C01814=1060.233,-44.337,-65.681,171.446,27.282,155.095
C01815=1060.228,-44.587,-65.669,171.444,27.280,155.095
C01816=1060.221,-44.836,-65.657,171.442,27.279,155.095
C01817=1060.215,-45.086,-65.644,171.441,27.277,155.095
C01818=1060.209,-45.335,-65.631,171.439,27.275,155.095
C01819=1060.203,-45.585,-65.619,171.437,27.273,155.094
C01820=1060.196,-45.835,-65.607,171.436,27.271,155.094
C01821=1060.190,-46.085,-65.594,171.434,27.269,155.094
C01822=1060.184,-46.335,-65.581,171.432,27.267,155.094
C01823=1060.178,-46.584,-65.568,171.431,27.265,155.094
C01824=1060.172,-46.833,-65.556,171.429,27.263,155.093
C01825=1060.166,-47.083,-65.544,171.428,27.261,155.093
C01826=1060.160,-47.332,-65.531,171.426,27.259,155.093
C01827=1060.154,-47.582,-65.519,171.424,27.257,155.093
C01828=1060.147,-47.831,-65.506,171.423,27.255,155.093
C01829=1060.142,-48.081,-65.494,171.421,27.254,155.093
C01830=1060.136,-48.331,-65.481,171.419,27.251,155.092
C01831=1060.130,-48.581,-65.469,171.418,27.250,155.092
C01832=1060.123,-48.831,-65.457,171.416,27.247,155.092
C01833=1060.117,-49.080,-65.444,171.414,27.246,155.092
C01834=1060.112,-49.330,-65.432,171.413,27.244,155.092
C01835=1060.105,-49.579,-65.419,171.411,27.242,155.091
C01836=1060.099,-49.828,-65.407,171.409,27.240,155.091
C01837=1060.093,-50.108,-65.393,171.408,27.238,155.091
C01838=1060.086,-50.387,-65.379,171.406,27.236,155.091
C01839=1060.078,-50.667,-65.365,171.403,27.234,155.091
C01840=1060.071,-50.946,-65.352,171.402,27.232,155.091
C01841=1060.065,-51.195,-65.340,171.400,27.230,155.090
C01842=1060.059,-51.444,-65.327,171.399,27.228,155.090
C01843=1060.053,-51.694,-65.315,171.397,27.227,155.090
C01844=1060.047,-51.944,-65.303,171.395,27.225,155.090
C01845=1060.040,-52.193,-65.291,171.394,27.223,155.090
C01846=1060.034,-52.443,-65.278,171.392,27.221,155.090
C01847=1060.028,-52.693,-65.266,171.390,27.219,155.089
C01848=1060.021,-52.942,-65.254,171.389,27.218,155.089
C01849=1060.015,-53.192,-65.242,171.387,27.216,155.089
C01850=1060.008,-53.442,-65.230,171.385,27.214,155.089
C01851=1060.003,-53.691,-65.218,171.384,27.213,155.089
C01852=1059.996,-53.941,-65.206,171.382,27.211,155.089
C01853=1059.990,-54.190,-65.194,171.380,27.209,155.089
C01854=1059.984,-54.440,-65.181,171.378,27.207,155.088
C01855=1059.977,-54.690,-65.169,171.377,27.206,155.088
C01856=1059.971,-54.940,-65.157,171.375,27.203,155.088
C01857=1059.965,-55.189,-65.145,171.374,27.202,155.088
C01858=1059.959,-55.438,-65.133,171.371,27.200,155.088
C01859=1059.953,-55.688,-65.121,171.369,27.198,155.088
C01860=1059.946,-55.938,-65.109,171.368,27.196,155.087
C01861=1059.940,-56.188,-65.097,171.366,27.195,155.087
C01862=1059.934,-56.437,-65.085,171.364,27.193,155.087
C01863=1059.928,-56.686,-65.073,171.362,27.191,155.087
C01864=1059.922,-56.936,-65.061,171.361,27.190,155.087
C01865=1059.915,-57.186,-65.049,171.359,27.188,155.087
C01866=1059.909,-57.435,-65.037,171.357,27.186,155.087
C01867=1059.903,-57.686,-65.025,171.356,27.184,155.086
C01868=1059.897,-57.935,-65.013,171.354,27.183,155.086
C01869=1059.890,-58.184,-65.001,171.352,27.181,155.086
C01870=1059.884,-58.434,-64.989,171.351,27.179,155.086
C01871=1059.878,-58.684,-64.977,171.349,27.178,155.086
C01872=1059.872,-58.933,-64.966,171.347,27.176,155.086
C01873=1059.866,-59.183,-64.953,171.346,27.174,155.086
C01874=1059.859,-59.433,-64.942,171.344,27.172,155.085
C01875=1059.853,-59.682,-64.930,171.342,27.171,155.085
C01876=1059.847,-59.931,-64.917,171.341,27.169,155.085
C01877=1059.841,-60.182,-64.906,171.339,27.167,155.085
C01878=1059.834,-60.431,-64.894,171.337,27.166,155.085
C01879=1059.829,-60.681,-64.882,171.336,27.164,155.085
C01880=1059.823,-60.930,-64.870,171.334,27.162,155.085
C01881=1059.816,-61.180,-64.859,171.332,27.161,155.084
C01882=1059.810,-61.430,-64.846,171.331,27.159,155.084
C01883=1059.804,-61.680,-64.834,171.329,27.157,155.084
C01884=1059.798,-61.929,-64.823,171.326,27.155,155.084
C01885=1059.792,-62.179,-64.811,171.325,27.153,155.084
C01886=1059.785,-62.429,-64.799,171.323,27.152,155.084
C01887=1059.779,-62.677,-64.787,171.321,27.150,155.084
C01888=1059.774,-62.928,-64.775,171.320,27.148,155.083
C01889=1059.767,-63.178,-64.763,171.318,27.147,155.083
C01890=1059.761,-63.426,-64.752,171.316,27.145,155.083
C01891=1059.755,-63.677,-64.740,171.315,27.143,155.083
C01892=1059.749,-63.926,-64.728,171.313,27.141,155.083
C01893=1059.743,-64.175,-64.717,171.311,27.140,155.083
C01894=1059.736,-64.426,-64.705,171.309,27.138,155.083
C01895=1059.730,-64.675,-64.693,171.308,27.136,155.082
C01896=1059.725,-64.925,-64.682,171.306,27.135,155.082
C01897=1059.718,-65.174,-64.670,171.304,27.134,155.082
C01898=1059.712,-65.424,-64.657,171.303,27.132,155.082
C01899=1059.706,-65.674,-64.646,171.301,27.130,155.082
C01900=1059.700,-65.923,-64.634,171.299,27.128,155.082
C01901=1059.693,-66.204,-64.622,171.297,27.126,155.082
C01902=1059.686,-66.484,-64.608,171.295,27.125,155.082
C01903=1059.680,-66.765,-64.596,171.293,27.123,155.081
C01904=1059.672,-67.045,-64.582,171.292,27.121,155.081
C01905=1059.667,-67.295,-64.571,171.290,27.120,155.081
C01906=1059.661,-67.545,-64.559,171.287,27.118,155.081
C01907=1059.654,-67.794,-64.547,171.286,27.116,155.081
C01908=1059.648,-68.044,-64.536,171.284,27.114,155.081
C01909=1059.642,-68.293,-64.523,171.282,27.112,155.081
C01910=1059.637,-68.543,-64.512,171.281,27.111,155.080
C01911=1059.630,-68.793,-64.501,171.279,27.109,155.080
C01912=1059.624,-69.042,-64.490,171.277,27.107,155.080
C01913=1059.618,-69.292,-64.477,171.276,27.106,155.080
C01914=1059.612,-69.542,-64.466,171.274,27.104,155.080
C01915=1059.606,-69.791,-64.454,171.272,27.103,155.080
C01916=1059.600,-70.041,-64.443,171.270,27.101,155.080
C01917=1059.594,-70.291,-64.432,171.269,27.099,155.080
C01918=1059.588,-70.541,-64.420,171.267,27.098,155.079
C01919=1059.582,-70.790,-64.409,171.265,27.097,155.079
C01920=1059.576,-71.040,-64.397,171.264,27.095,155.079
C01921=1059.570,-71.289,-64.386,171.262,27.093,155.079
C01922=1059.564,-71.539,-64.373,171.260,27.091,155.079
C01923=1059.558,-71.788,-64.362,171.259,27.090,155.079
C01924=1059.552,-72.039,-64.351,171.257,27.089,155.079
C01925=1059.546,-72.288,-64.340,171.255,27.087,155.079
C01926=1059.539,-72.538,-64.328,171.253,27.085,155.079
C01927=1059.534,-72.787,-64.316,171.251,27.083,155.078
C01928=1059.528,-73.037,-64.305,171.249,27.082,155.078
C01929=1059.522,-73.287,-64.294,171.247,27.080,155.078
C01930=1059.515,-73.536,-64.282,171.246,27.079,155.078
C01931=1059.510,-73.786,-64.271,171.244,27.077,155.078
C01932=1059.504,-74.036,-64.259,171.242,27.076,155.078
C01933=1059.497,-74.285,-64.248,171.241,27.074,155.078
C01934=1059.491,-74.535,-64.237,171.239,27.072,155.078
C01935=1059.485,-74.784,-64.226,171.237,27.071,155.078
C01936=1059.479,-75.034,-64.214,171.235,27.070,155.078
C01937=1059.473,-75.283,-64.203,171.234,27.068,155.077
C01938=1059.467,-75.534,-64.192,171.232,27.067,155.077
C01939=1059.461,-75.783,-64.181,171.230,27.065,155.077
C01940=1059.454,-76.033,-64.169,171.229,27.064,155.077
C01941=1059.448,-76.282,-64.158,171.227,27.062,155.077
C01942=1059.442,-76.532,-64.147,171.225,27.061,155.077
C01943=1059.436,-76.782,-64.136,171.223,27.059,155.077
C01944=1059.430,-77.031,-64.124,171.221,27.057,155.077
C01945=1059.424,-77.281,-64.113,171.219,27.056,155.077
C01946=1059.418,-77.531,-64.102,171.217,27.054,155.077
C01947=1059.412,-77.781,-64.091,171.216,27.053,155.077
C01948=1059.406,-78.031,-64.080,171.214,27.052,155.076
C01949=1059.399,-78.280,-64.069,171.212,27.051,155.076
C01950=1059.393,-78.530,-64.057,171.210,27.049,155.076
C01951=1059.387,-78.779,-64.046,171.209,27.048,155.076
C01952=1059.381,-79.030,-64.035,171.207,27.046,155.076
C01953=1059.375,-79.279,-64.024,171.205,27.045,155.076
C01954=1059.369,-79.528,-64.013,171.204,27.043,155.076
C01955=1059.363,-79.778,-64.001,171.202,27.042,155.076
C01956=1059.356,-80.027,-63.991,171.200,27.040,155.076
C01957=1059.350,-80.277,-63.980,171.198,27.039,155.076
C01958=1059.344,-80.527,-63.969,171.196,27.037,155.076
C01959=1059.338,-80.777,-63.958,171.194,27.036,155.076
C01960=1059.332,-81.026,-63.948,171.192,27.035,155.076
C01961=1059.325,-81.277,-63.936,171.191,27.033,155.075
C01962=1059.319,-81.526,-63.925,171.189,27.032,155.075
C01963=1059.312,-81.776,-63.915,171.187,27.031,155.075
C01964=1059.306,-82.025,-63.903,171.185,27.029,155.075
C01965=1059.300,-82.308,-63.891,171.183,27.028,155.075
C01966=1059.292,-82.590,-63.878,171.181,27.026,155.075
C01967=1059.285,-82.873,-63.867,171.179,27.025,155.075
C01968=1059.279,-83.156,-63.854,171.177,27.023,155.075
C01969=1059.272,-83.405,-63.844,171.176,27.022,155.075
C01970=1059.266,-83.655,-63.832,171.173,27.021,155.075
C01971=1059.260,-83.905,-63.821,171.171,27.019,155.075
C01972=1059.254,-84.154,-63.811,171.169,27.018,155.075
C01973=1059.247,-84.404,-63.800,171.168,27.017,155.075
C01974=1059.241,-84.654,-63.789,171.166,27.015,155.075
C01975=1059.235,-84.904,-63.778,171.164,27.014,155.075
C01976=1059.229,-85.153,-63.767,171.162,27.013,155.075
C01977=1059.223,-85.403,-63.757,171.161,27.012,155.075
C01978=1059.216,-85.653,-63.745,171.159,27.010,155.074
C01979=1059.210,-85.902,-63.735,171.157,27.009,155.074
C01980=1059.204,-86.152,-63.724,171.155,27.008,155.074
C01981=1059.198,-86.402,-63.713,171.154,27.007,155.074
C01982=1059.191,-86.651,-63.703,171.152,27.005,155.074
C01983=1059.185,-86.901,-63.691,171.149,27.004,155.074
C01984=1059.179,-87.151,-63.681,171.148,27.002,155.074
C01985=1059.173,-87.400,-63.670,171.146,27.001,155.074
C01986=1059.167,-87.651,-63.660,171.144,27.000,155.074
C01987=1059.161,-87.900,-63.649,171.142,26.998,155.074
C01988=1059.155,-88.149,-63.639,171.141,26.997,155.074
C01989=1059.148,-88.399,-63.627,171.139,26.996,155.074
C01990=1059.143,-88.649,-63.616,171.137,26.994,155.074
C01991=1059.136,-88.898,-63.606,171.135,26.993,155.074
C01992=1059.130,-89.148,-63.595,171.134,26.992,155.074
C01993=1059.124,-89.398,-63.585,171.132,26.991,155.074
C01994=1059.118,-89.648,-63.574,171.130,26.990,155.074
C01995=1059.112,-89.897,-63.564,171.128,26.989,155.074
C01996=1059.106,-90.147,-63.552,171.126,26.987,155.074
C01997=1059.099,-90.396,-63.542,171.124,26.986,155.074
C01998=1059.094,-90.646,-63.531,171.122,26.985,155.074
C01999=1059.087,-90.896,-63.521,171.120,26.983,155.074
C02000=1059.081,-91.146,-63.510,171.118,26.982,155.074
C02001=1059.075,-91.395,-63.500,171.117,26.981,155.074
C02002=1059.069,-91.645,-63.489,171.115,26.980,155.073
C02003=1059.063,-91.895,-63.479,171.113,26.978,155.073
C02004=1059.057,-92.145,-63.468,171.111,26.977,155.073
C02005=1059.051,-92.394,-63.458,171.110,26.976,155.073
C02006=1059.045,-92.644,-63.447,171.108,26.975,155.073
C02007=1059.038,-92.894,-63.437,171.106,26.974,155.073
C02008=1059.032,-93.144,-63.426,171.104,26.973,155.073
C02009=1059.027,-93.393,-63.415,171.102,26.971,155.073
C02010=1059.020,-93.642,-63.405,171.100,26.970,155.073
C02011=1059.014,-93.893,-63.394,171.098,26.969,155.073
C02012=1059.008,-94.142,-63.384,171.096,26.967,155.073
C02013=1059.002,-94.392,-63.373,171.095,26.966,155.073
C02014=1058.996,-94.642,-63.363,171.093,26.965,155.073
C02015=1058.990,-94.891,-63.353,171.091,26.964,155.073
C02016=1058.984,-95.141,-63.341,171.089,26.963,155.073
C02017=1058.977,-95.391,-63.332,171.088,26.962,155.073
C02018=1058.972,-95.640,-63.321,171.086,26.961,155.073
C02019=1058.966,-95.890,-63.310,171.084,26.959,155.073
C02020=1058.960,-96.140,-63.300,171.082,26.958,155.073
C02021=1058.954,-96.389,-63.290,171.079,26.957,155.073
C02022=1058.947,-96.639,-63.279,171.078,26.956,155.073
C02023=1058.942,-96.889,-63.269,171.076,26.955,155.073
C02024=1058.935,-97.138,-63.258,171.074,26.954,155.073
C02025=1058.930,-97.388,-63.248,171.072,26.952,155.073
C02026=1058.923,-97.638,-63.238,171.071,26.951,155.073
C02027=1058.917,-97.887,-63.227,171.069,26.950,155.073
C02028=1058.911,-98.138,-63.217,171.067,26.949,155.073
C02029=1058.904,-98.422,-63.205,171.065,26.948,155.073
C02030=1058.897,-98.707,-63.193,171.063,26.947,155.073
C02031=1058.889,-98.993,-63.182,171.061,26.945,155.073
C02032=1058.883,-99.277,-63.170,171.058,26.944,155.073
C02033=1058.876,-99.526,-63.160,171.056,26.943,155.073
C02034=1058.871,-99.777,-63.150,171.055,26.942,155.073
C02035=1058.864,-100.026,-63.140,171.053,26.941,155.073
C02036=1058.858,-100.276,-63.130,171.051,26.939,155.073
C02037=1058.852,-100.526,-63.119,171.049,26.939,155.073
C02038=1058.846,-100.776,-63.109,171.047,26.938,155.073
C02039=1058.839,-101.025,-63.099,171.046,26.937,155.073
C02040=1058.834,-101.275,-63.089,171.044,26.936,155.073
C02041=1058.827,-101.524,-63.079,171.042,26.934,155.073
C02042=1058.821,-101.774,-63.069,171.040,26.934,155.073
C02043=1058.815,-102.025,-63.058,171.037,26.933,155.073
C02044=1058.809,-102.274,-63.048,171.036,26.931,155.073
C02045=1058.802,-102.524,-63.039,171.034,26.930,155.073
C02046=1058.797,-102.773,-63.028,171.032,26.929,155.073
C02047=1058.790,-103.023,-63.018,171.030,26.929,155.073
C02048=1058.784,-103.272,-63.008,171.028,26.927,155.073
C02049=1058.779,-103.522,-62.998,171.027,26.926,155.073
C02050=1058.772,-103.772,-62.988,171.025,26.925,155.073
C02051=1058.766,-104.021,-62.978,171.023,26.925,155.073
C02052=1058.760,-104.272,-62.967,171.021,26.924,155.073
C02053=1058.754,-104.522,-62.958,171.019,26.922,155.073
C02054=1058.747,-104.771,-62.948,171.018,26.922,155.073
C02055=1058.741,-105.021,-62.938,171.015,26.920,155.073
C02056=1058.735,-105.270,-62.927,171.013,26.919,155.073
C02057=1058.729,-105.520,-62.918,171.011,26.918,155.073
C02058=1058.723,-105.770,-62.908,171.009,26.918,155.073
C02059=1058.716,-106.019,-62.898,171.008,26.917,155.073
C02060=1058.711,-106.269,-62.887,171.006,26.915,155.073
C02061=1058.705,-106.519,-62.878,171.004,26.915,155.073
C02062=1058.699,-106.769,-62.868,171.002,26.914,155.073
C02063=1058.692,-107.018,-62.858,171.000,26.913,155.073
C02064=1058.687,-107.268,-62.848,170.999,26.912,155.073
C02065=1058.681,-107.518,-62.838,170.997,26.911,155.073
C02066=1058.674,-107.767,-62.828,170.994,26.910,155.073
C02067=1058.668,-108.017,-62.818,170.992,26.909,155.073
C02068=1058.661,-108.267,-62.809,170.990,26.908,155.073
C02069=1058.655,-108.517,-62.799,170.989,26.907,155.073
C02070=1058.649,-108.766,-62.789,170.987,26.906,155.073
C02071=1058.643,-109.016,-62.779,170.985,26.906,155.073
C02072=1058.637,-109.266,-62.769,170.983,26.905,155.073
C02073=1058.631,-109.516,-62.759,170.981,26.904,155.073
C02074=1058.625,-109.766,-62.750,170.979,26.903,155.073
C02075=1058.618,-110.015,-62.740,170.978,26.902,155.074
C02076=1058.612,-110.265,-62.730,170.976,26.901,155.073
C02077=1058.606,-110.514,-62.720,170.973,26.900,155.074
C02078=1058.600,-110.764,-62.711,170.971,26.899,155.074
C02079=1058.594,-111.014,-62.701,170.969,26.899,155.074
C02080=1058.588,-111.264,-62.691,170.968,26.898,155.074
C02081=1058.582,-111.513,-62.681,170.966,26.897,155.074
C02082=1058.575,-111.763,-62.671,170.964,26.896,155.074
C02083=1058.569,-112.013,-62.662,170.962,26.895,155.074
C02084=1058.563,-112.263,-62.652,170.960,26.894,155.074
C02085=1058.557,-112.513,-62.643,170.958,26.894,155.074
C02086=1058.551,-112.762,-62.633,170.957,26.893,155.074
C02087=1058.544,-113.012,-62.623,170.955,26.892,155.074
C02088=1058.538,-113.262,-62.614,170.953,26.891,155.074
C02089=1058.532,-113.511,-62.604,170.950,26.890,155.074
C02090=1058.526,-113.761,-62.593,170.948,26.890,155.074
C02091=1058.520,-114.011,-62.584,170.946,26.889,155.074
C02092=1058.515,-114.260,-62.575,170.945,26.888,155.074
C02093=1058.507,-114.543,-62.564,170.943,26.887,155.074
C02094=1058.500,-114.827,-62.553,170.940,26.886,155.074
C02095=1058.493,-115.111,-62.542,170.938,26.886,155.075
C02096=1058.486,-115.394,-62.531,170.936,26.884,155.074
C02097=1058.480,-115.644,-62.522,170.934,26.884,155.075
C02098=1058.474,-115.894,-62.512,170.933,26.883,155.075
C02099=1058.468,-116.144,-62.503,170.930,26.882,155.075
C02100=1058.462,-116.393,-62.493,170.928,26.881,155.075
C02101=1058.456,-116.643,-62.484,170.926,26.881,155.075
C02102=1058.450,-116.892,-62.474,170.924,26.880,155.075
C02103=1058.443,-117.142,-62.465,170.922,26.879,155.075
C02104=1058.437,-117.392,-62.456,170.920,26.879,155.075
C02105=1058.431,-117.641,-62.446,170.919,26.878,155.075
C02106=1058.425,-117.891,-62.437,170.917,26.877,155.075
C02107=1058.418,-118.141,-62.427,170.915,26.876,155.075
C02108=1058.412,-118.391,-62.418,170.913,26.876,155.075
C02109=1058.406,-118.641,-62.408,170.911,26.875,155.075
C02110=1058.400,-118.890,-62.398,170.908,26.874,155.075
C02111=1058.394,-119.140,-62.389,170.907,26.873,155.076
C02112=1058.388,-119.390,-62.379,170.905,26.873,155.076
C02113=1058.382,-119.639,-62.370,170.903,26.872,155.076
C02114=1058.376,-119.889,-62.361,170.901,26.871,155.076
C02115=1058.369,-120.139,-62.352,170.899,26.871,155.076
C02116=1058.363,-120.389,-62.343,170.897,26.870,155.076
C02117=1058.357,-120.639,-62.333,170.895,26.870,155.076
C02118=1058.351,-120.888,-62.324,170.894,26.868,155.076
C02119=1058.345,-121.138,-62.314,170.892,26.868,155.076
C02120=1058.339,-121.387,-62.305,170.890,26.867,155.076
C02121=1058.333,-121.637,-62.295,170.888,26.867,155.076
C02122=1058.327,-121.888,-62.286,170.885,26.866,155.076
C02123=1058.320,-122.137,-62.277,170.883,26.866,155.077
C02124=1058.314,-122.387,-62.268,170.881,26.865,155.077
C02125=1058.308,-122.637,-62.258,170.880,26.864,155.077
C02126=1058.302,-122.886,-62.249,170.878,26.863,155.077
C02127=1058.296,-123.136,-62.240,170.876,26.863,155.077
C02128=1058.290,-123.386,-62.231,170.874,26.862,155.077
C02129=1058.283,-123.635,-62.222,170.872,26.862,155.077
C02130=1058.277,-123.885,-62.212,170.870,26.861,155.077
C02131=1058.271,-124.135,-62.203,170.868,26.861,155.077
C02132=1058.266,-124.385,-62.194,170.866,26.860,155.077
C02133=1058.259,-124.635,-62.184,170.864,26.859,155.077
C02134=1058.252,-124.884,-62.176,170.862,26.859,155.078
C02135=1058.246,-125.134,-62.166,170.860,26.858,155.078
C02136=1058.240,-125.384,-62.157,170.858,26.858,155.078
C02137=1058.235,-125.633,-62.148,170.856,26.857,155.078
C02138=1058.228,-125.883,-62.139,170.854,26.857,155.078
C02139=1058.222,-126.133,-62.130,170.852,26.856,155.078
C02140=1058.216,-126.383,-62.120,170.850,26.856,155.078
C02141=1058.210,-126.633,-62.111,170.849,26.855,155.078
C02142=1058.204,-126.882,-62.103,170.847,26.855,155.078
C02143=1058.198,-127.132,-62.093,170.845,26.854,155.078
C02144=1058.191,-127.382,-62.084,170.843,26.853,155.078
C02145=1058.185,-127.632,-62.076,170.840,26.853,155.079
C02146=1058.179,-127.882,-62.066,170.838,26.852,155.079
C02147=1058.174,-128.131,-62.056,170.836,26.851,155.079
C02148=1058.171,-128.382,-62.046,170.835,26.849,155.079
C02149=1058.168,-128.632,-62.034,170.833,26.847,155.078
C02150=1058.168,-128.883,-62.023,170.833,26.844,155.078
C02151=1058.169,-129.133,-62.010,170.831,26.841,155.078
C02152=1058.170,-129.383,-61.997,170.830,26.837,155.077
C02153=1058.173,-129.635,-61.983,170.830,26.833,155.076
C02154=1058.177,-129.886,-61.968,170.829,26.827,155.075
C02155=1058.183,-130.137,-61.952,170.828,26.822,155.075
C02156=1058.190,-130.387,-61.937,170.828,26.816,155.073
C02157=1057.814,-130.410,-62.137,170.780,26.978,155.107
C02158=1057.807,-130.160,-62.154,170.781,26.984,155.108
C02159=1057.802,-129.909,-62.169,170.781,26.990,155.109
C02160=1057.797,-129.658,-62.183,170.782,26.995,155.109
C02161=1057.794,-129.406,-62.197,170.782,26.999,155.110
C02162=1057.791,-129.156,-62.211,170.783,27.003,155.111
C02163=1057.791,-128.906,-62.224,170.785,27.006,155.111
C02164=1057.792,-128.656,-62.236,170.786,27.009,155.112
C02165=1057.795,-128.405,-62.246,170.788,27.012,155.112
C02166=1057.798,-128.155,-62.257,170.789,27.013,155.112
C02167=1057.803,-127.905,-62.267,170.791,27.015,155.112
C02168=1057.809,-127.655,-62.276,170.793,27.015,155.112
C02169=1057.815,-127.405,-62.286,170.795,27.016,155.112
C02170=1057.821,-127.154,-62.295,170.797,27.016,155.112
C02171=1057.826,-126.905,-62.304,170.799,27.017,155.112
C02172=1057.833,-126.656,-62.313,170.801,27.017,155.111
C02173=1057.839,-126.405,-62.322,170.803,27.018,155.111
C02174=1057.845,-126.156,-62.331,170.804,27.018,155.111
C02175=1057.852,-125.906,-62.340,170.806,27.019,155.111
C02176=1057.858,-125.656,-62.349,170.808,27.019,155.111
C02177=1057.864,-125.407,-62.358,170.810,27.020,155.111
C02178=1057.870,-125.157,-62.368,170.813,27.021,155.111
C02179=1057.877,-124.907,-62.377,170.815,27.021,155.111
C02180=1057.883,-124.657,-62.386,170.817,27.022,155.111
C02181=1057.888,-124.408,-62.395,170.819,27.022,155.111
C02182=1057.894,-124.158,-62.404,170.820,27.023,155.110
C02183=1057.901,-123.909,-62.413,170.822,27.023,155.110
C02184=1057.907,-123.658,-62.422,170.824,27.024,155.110
C02185=1057.913,-123.408,-62.432,170.826,27.024,155.110
C02186=1057.919,-123.159,-62.441,170.828,27.025,155.110
C02187=1057.925,-122.910,-62.450,170.830,27.025,155.110
C02188=1057.931,-122.660,-62.460,170.832,27.026,155.110
C02189=1057.938,-122.410,-62.468,170.835,27.027,155.110
C02190=1057.944,-122.160,-62.478,170.836,27.028,155.110
C02191=1057.950,-121.910,-62.487,170.838,27.028,155.110
C02192=1057.956,-121.661,-62.497,170.840,27.029,155.110
C02193=1057.962,-121.411,-62.506,170.842,27.029,155.109
C02194=1057.968,-121.161,-62.515,170.844,27.030,155.109
C02195=1057.974,-120.911,-62.525,170.846,27.030,155.109
C02196=1057.980,-120.661,-62.534,170.848,27.031,155.109
C02197=1057.987,-120.412,-62.543,170.849,27.032,155.109
C02198=1057.993,-120.162,-62.553,170.851,27.033,155.109
C02199=1057.999,-119.912,-62.562,170.853,27.033,155.109
C02200=1058.005,-119.663,-62.571,170.856,27.034,155.109
C02201=1058.011,-119.413,-62.581,170.858,27.034,155.109
C02202=1058.017,-119.163,-62.591,170.860,27.035,155.109
C02203=1058.023,-118.913,-62.599,170.862,27.036,155.109
C02204=1058.029,-118.663,-62.609,170.863,27.037,155.109
C02205=1058.036,-118.413,-62.619,170.865,27.037,155.109
C02206=1058.042,-118.164,-62.628,170.867,27.038,155.109
C02207=1058.049,-117.914,-62.637,170.869,27.039,155.108
C02208=1058.055,-117.664,-62.647,170.871,27.039,155.108
C02209=1058.060,-117.415,-62.656,170.873,27.040,155.108
C02210=1058.067,-117.165,-62.665,170.875,27.041,155.108
C02211=1058.073,-116.916,-62.675,170.877,27.042,155.108
C02212=1058.079,-116.666,-62.685,170.879,27.042,155.108
C02213=1058.085,-116.416,-62.694,170.881,27.043,155.108
C02214=1058.091,-116.166,-62.704,170.883,27.044,155.108
C02215=1058.097,-115.916,-62.713,170.885,27.044,155.108
C02216=1058.104,-115.667,-62.723,170.887,27.045,155.108
C02217=1058.110,-115.417,-62.732,170.888,27.046,155.108
C02218=1058.117,-115.133,-62.743,170.891,27.047,155.108
C02219=1058.123,-114.850,-62.754,170.893,27.047,155.108
C02220=1058.131,-114.566,-62.765,170.895,27.048,155.108
C02221=1058.138,-114.283,-62.776,170.898,27.049,155.107
C02222=1058.143,-114.034,-62.785,170.900,27.050,155.107
C02223=1058.150,-113.784,-62.795,170.901,27.051,155.107
C02224=1058.156,-113.535,-62.805,170.903,27.051,155.107
C02225=1058.162,-113.285,-62.814,170.905,27.053,155.107
C02226=1058.168,-113.035,-62.824,170.907,27.053,155.107
C02227=1058.174,-112.785,-62.834,170.909,27.054,155.107
C02228=1058.180,-112.535,-62.844,170.911,27.055,155.107
C02229=1058.186,-112.285,-62.853,170.912,27.056,155.107
C02230=1058.192,-112.035,-62.863,170.915,27.057,155.107
C02231=1058.199,-111.786,-62.872,170.917,27.058,155.107
C02232=1058.205,-111.536,-62.883,170.919,27.058,155.107
C02233=1058.211,-111.287,-62.892,170.921,27.059,155.107
C02234=1058.217,-111.037,-62.902,170.923,27.060,155.107
C02235=1058.224,-110.787,-62.911,170.924,27.061,155.107
C02236=1058.230,-110.537,-62.921,170.926,27.062,155.107
C02237=1058.235,-110.287,-62.931,170.928,27.062,155.107
C02238=1058.242,-110.038,-62.941,170.930,27.063,155.107
C02239=1058.248,-109.788,-62.951,170.932,27.064,155.107
C02240=1058.254,-109.538,-62.960,170.934,27.065,155.107
C02241=1058.260,-109.289,-62.970,170.936,27.066,155.107
C02242=1058.266,-109.039,-62.980,170.938,27.067,155.107
C02243=1058.273,-108.790,-62.990,170.940,27.068,155.107
C02244=1058.279,-108.540,-62.999,170.942,27.068,155.106
C02245=1058.284,-108.290,-63.010,170.944,27.070,155.107
C02246=1058.291,-108.039,-63.020,170.946,27.070,155.106
C02247=1058.298,-107.790,-63.030,170.947,27.071,155.106
C02248=1058.304,-107.540,-63.039,170.949,27.072,155.106
C02249=1058.310,-107.290,-63.049,170.951,27.073,155.106
C02250=1058.316,-107.041,-63.059,170.953,27.074,155.106
C02251=1058.322,-106.791,-63.069,170.955,27.075,155.106
C02252=1058.328,-106.541,-63.079,170.957,27.076,155.106
C02253=1058.334,-106.292,-63.089,170.959,27.077,155.106
C02254=1058.341,-106.042,-63.099,170.961,27.078,155.106
C02255=1058.346,-105.792,-63.109,170.963,27.079,155.106
C02256=1058.352,-105.542,-63.119,170.965,27.080,155.106
C02257=1058.359,-105.293,-63.129,170.966,27.080,155.106
C02258=1058.365,-105.043,-63.138,170.968,27.081,155.106
C02259=1058.370,-104.793,-63.149,170.970,27.083,155.106
C02260=1058.377,-104.544,-63.159,170.972,27.083,155.106
C02261=1058.383,-104.294,-63.168,170.974,27.084,155.106
C02262=1058.389,-104.044,-63.179,170.975,27.085,155.106
C02263=1058.396,-103.794,-63.189,170.978,27.086,155.106
C02264=1058.402,-103.545,-63.199,170.980,27.087,155.106
C02265=1058.408,-103.295,-63.209,170.982,27.088,155.106
C02266=1058.414,-103.045,-63.219,170.984,27.089,155.106
C02267=1058.420,-102.796,-63.229,170.986,27.090,155.106
C02268=1058.426,-102.546,-63.239,170.987,27.091,155.106
C02269=1058.432,-102.296,-63.249,170.989,27.092,155.106
C02270=1058.438,-102.047,-63.260,170.991,27.093,155.106
C02271=1058.445,-101.797,-63.269,170.993,27.094,155.106
C02272=1058.451,-101.547,-63.280,170.995,27.095,155.106
C02273=1058.457,-101.297,-63.290,170.996,27.096,155.106
C02274=1058.463,-101.048,-63.300,170.999,27.098,155.106
C02275=1058.469,-100.798,-63.310,171.001,27.099,155.106
C02276=1058.475,-100.549,-63.321,171.003,27.100,155.106
C02277=1058.481,-100.299,-63.330,171.005,27.100,155.106
C02278=1058.488,-100.049,-63.341,171.006,27.101,155.106
C02279=1058.494,-99.799,-63.351,171.008,27.103,155.106
C02280=1058.500,-99.550,-63.361,171.010,27.104,155.106
C02281=1058.506,-99.300,-63.371,171.012,27.105,155.106
C02282=1058.513,-99.015,-63.383,171.014,27.106,155.106
C02283=1058.520,-98.729,-63.394,171.016,27.107,155.106
C02284=1058.527,-98.445,-63.406,171.018,27.108,155.106
C02285=1058.534,-98.159,-63.419,171.021,27.110,155.106
C02286=1058.541,-97.910,-63.428,171.023,27.110,155.106
C02287=1058.547,-97.660,-63.438,171.024,27.111,155.106
C02288=1058.553,-97.411,-63.449,171.026,27.113,155.106
C02289=1058.559,-97.161,-63.459,171.028,27.114,155.106
C02290=1058.565,-96.912,-63.470,171.030,27.115,155.106
C02291=1058.571,-96.661,-63.480,171.031,27.116,155.106
C02292=1058.577,-96.412,-63.491,171.033,27.117,155.106
C02293=1058.583,-96.162,-63.501,171.035,27.118,155.106
C02294=1058.589,-95.912,-63.511,171.037,27.119,155.106
C02295=1058.595,-95.663,-63.522,171.040,27.121,155.106
C02296=1058.602,-95.413,-63.533,171.041,27.122,155.106
C02297=1058.607,-95.163,-63.543,171.043,27.123,155.106
C02298=1058.613,-94.913,-63.554,171.045,27.125,155.106
C02299=1058.620,-94.664,-63.564,171.047,27.126,155.106
C02300=1058.625,-94.414,-63.574,171.048,27.127,155.106
C02301=1058.632,-94.164,-63.585,171.050,27.128,155.106
C02302=1058.638,-93.915,-63.596,171.052,27.129,155.106
C02303=1058.643,-93.665,-63.606,171.054,27.130,155.106
C02304=1058.650,-93.415,-63.616,171.055,27.131,155.106
C02305=1058.656,-93.166,-63.627,171.057,27.132,155.106
C02306=1058.663,-92.916,-63.638,171.059,27.134,155.106
C02307=1058.668,-92.666,-63.648,171.062,27.135,155.106
C02308=1058.674,-92.417,-63.659,171.064,27.136,155.106
C02309=1058.680,-92.167,-63.669,171.065,27.138,155.107
C02310=1058.687,-91.917,-63.680,171.067,27.139,155.107
C02311=1058.692,-91.667,-63.690,171.069,27.140,155.107
C02312=1058.699,-91.418,-63.701,171.071,27.141,155.107
C02313=1058.704,-91.168,-63.711,171.072,27.142,155.107
C02314=1058.711,-90.918,-63.722,171.074,27.143,155.107
C02315=1058.717,-90.668,-63.732,171.076,27.144,155.107
C02316=1058.723,-90.419,-63.743,171.078,27.146,155.107
C02317=1058.730,-90.169,-63.754,171.079,27.147,155.107
C02318=1058.735,-89.920,-63.765,171.081,27.148,155.107
C02319=1058.741,-89.670,-63.776,171.084,27.150,155.107
C02320=1058.748,-89.421,-63.786,171.086,27.151,155.107
C02321=1058.754,-89.170,-63.796,171.087,27.152,155.107
C02322=1058.759,-88.921,-63.807,171.089,27.154,155.107
C02323=1058.766,-88.671,-63.817,171.091,27.155,155.107
C02324=1058.772,-88.421,-63.829,171.093,27.156,155.107
C02325=1058.778,-88.172,-63.840,171.094,27.157,155.107
C02326=1058.784,-87.923,-63.850,171.096,27.158,155.107
C02327=1058.791,-87.672,-63.861,171.098,27.160,155.107
C02328=1058.797,-87.423,-63.871,171.100,27.161,155.107
C02329=1058.803,-87.173,-63.882,171.101,27.162,155.107
C02330=1058.809,-86.923,-63.893,171.103,27.163,155.107
C02331=1058.815,-86.673,-63.904,171.105,27.165,155.108
C02332=1058.821,-86.424,-63.914,171.108,27.166,155.108
C02333=1058.828,-86.174,-63.925,171.109,27.167,155.108
C02334=1058.833,-85.924,-63.936,171.111,27.169,155.108
C02335=1058.840,-85.675,-63.947,171.113,27.170,155.108
C02336=1058.846,-85.425,-63.958,171.115,27.171,155.108
C02337=1058.852,-85.176,-63.969,171.116,27.173,155.108
C02338=1058.859,-84.926,-63.979,171.118,27.174,155.108
C02339=1058.865,-84.676,-63.990,171.120,27.175,155.108
C02340=1058.870,-84.427,-64.001,171.122,27.176,155.108
C02341=1058.877,-84.177,-64.012,171.124,27.178,155.108
C02342=1058.883,-83.927,-64.022,171.125,27.179,155.108
C02343=1058.890,-83.677,-64.034,171.127,27.180,155.108
C02344=1058.895,-83.428,-64.045,171.130,27.182,155.108
C02345=1058.902,-83.178,-64.055,171.131,27.183,155.108
C02346=1058.909,-82.895,-64.068,171.133,27.185,155.108
C02347=1058.916,-82.613,-64.080,171.135,27.186,155.108
C02348=1058.923,-82.331,-64.092,171.138,27.188,155.108
C02349=1058.930,-82.047,-64.104,171.139,27.189,155.108
C02350=1058.936,-81.798,-64.116,171.141,27.191,155.109
C02351=1058.943,-81.548,-64.126,171.143,27.192,155.109
C02352=1058.949,-81.298,-64.138,171.145,27.193,155.109
C02353=1058.955,-81.049,-64.149,171.146,27.194,155.109
C02354=1058.962,-80.799,-64.159,171.148,27.196,155.109
C02355=1058.968,-80.549,-64.170,171.150,27.197,155.109
C02356=1058.974,-80.299,-64.181,171.152,27.199,155.109
C02357=1058.980,-80.050,-64.192,171.154,27.200,155.109
C02358=1058.987,-79.800,-64.203,171.156,27.201,155.109
C02359=1058.992,-79.550,-64.214,171.158,27.203,155.109
C02360=1058.999,-79.301,-64.226,171.160,27.204,155.109
C02361=1059.005,-79.051,-64.237,171.161,27.205,155.109
C02362=1059.011,-78.802,-64.247,171.163,27.207,155.109
C02363=1059.017,-78.552,-64.259,171.165,27.208,155.109
C02364=1059.023,-78.302,-64.270,171.166,27.209,155.109
C02365=1059.029,-78.053,-64.282,171.168,27.211,155.110
C02366=1059.035,-77.803,-64.292,171.170,27.213,155.110
C02367=1059.041,-77.553,-64.304,171.172,27.214,155.110
C02368=1059.047,-77.303,-64.315,171.173,27.216,155.110
C02369=1059.054,-77.053,-64.326,171.175,27.217,155.110
C02370=1059.060,-76.804,-64.337,171.178,27.219,155.110
C02371=1059.066,-76.554,-64.349,171.179,27.220,155.110
C02372=1059.072,-76.305,-64.359,171.181,27.222,155.110
C02373=1059.078,-76.054,-64.371,171.183,27.223,155.110
C02374=1059.084,-75.806,-64.382,171.185,27.224,155.110
C02375=1059.090,-75.555,-64.394,171.186,27.226,155.111
C02376=1059.096,-75.306,-64.404,171.188,27.227,155.111
C02377=1059.103,-75.056,-64.416,171.190,27.229,155.111
C02378=1059.108,-74.807,-64.427,171.192,27.230,155.111
C02379=1059.115,-74.557,-64.439,171.193,27.232,155.111
C02380=1059.121,-74.307,-64.449,171.195,27.233,155.111
C02381=1059.127,-74.058,-64.461,171.197,27.235,155.111
C02382=1059.133,-73.808,-64.472,171.198,27.236,155.111
C02383=1059.139,-73.558,-64.483,171.200,27.238,155.111
C02384=1059.145,-73.309,-64.495,171.202,27.239,155.111
C02385=1059.152,-73.059,-64.506,171.204,27.241,155.111
C02386=1059.157,-72.809,-64.517,171.206,27.243,155.112
C02387=1059.163,-72.559,-64.530,171.208,27.244,155.112
C02388=1059.169,-72.310,-64.541,171.210,27.246,155.112
C02389=1059.176,-72.060,-64.553,171.211,27.247,155.112
C02390=1059.181,-71.811,-64.563,171.213,27.249,155.112
C02391=1059.188,-71.561,-64.575,171.215,27.251,155.112
C02392=1059.193,-71.312,-64.587,171.216,27.252,155.112
C02393=1059.199,-71.061,-64.598,171.218,27.253,155.112
C02394=1059.205,-70.813,-64.610,171.220,27.255,155.112
C02395=1059.212,-70.562,-64.621,171.222,27.257,155.113
C02396=1059.217,-70.313,-64.633,171.223,27.259,155.113
C02397=1059.223,-70.063,-64.644,171.225,27.260,155.113
C02398=1059.230,-69.813,-64.656,171.227,27.261,155.113
C02399=1059.236,-69.564,-64.667,171.228,27.263,155.113
C02400=1059.243,-69.314,-64.679,171.230,27.265,155.113
C02401=1059.248,-69.064,-64.691,171.232,27.266,155.113
C02402=1059.254,-68.815,-64.703,171.233,27.268,155.114
C02403=1059.260,-68.565,-64.714,171.235,27.270,155.114
C02404=1059.267,-68.316,-64.725,171.237,27.271,155.114
C02405=1059.272,-68.065,-64.737,171.239,27.273,155.114
C02406=1059.278,-67.816,-64.749,171.241,27.275,155.114
C02407=1059.285,-67.566,-64.760,171.243,27.276,155.114
C02408=1059.291,-67.317,-64.772,171.245,27.278,155.114
C02409=1059.296,-67.067,-64.784,171.246,27.280,155.114
C02410=1059.303,-66.787,-64.797,171.248,27.281,155.115
C02411=1059.310,-66.506,-64.809,171.250,27.283,155.115
C02412=1059.317,-66.226,-64.823,171.252,27.285,155.115
C02413=1059.324,-65.945,-64.836,171.254,27.287,155.115
C02414=1059.330,-65.696,-64.848,171.256,27.289,155.115
C02415=1059.335,-65.446,-64.859,171.257,27.290,155.115
C02416=1059.342,-65.196,-64.871,171.259,27.292,155.115
C02417=1059.349,-64.947,-64.883,171.261,27.294,155.115
C02418=1059.354,-64.697,-64.894,171.262,27.295,155.116
C02419=1059.360,-64.447,-64.907,171.264,27.296,155.116
C02420=1059.367,-64.197,-64.918,171.266,27.298,155.116
C02421=1059.373,-63.948,-64.930,171.268,27.300,155.116
C02422=1059.378,-63.698,-64.942,171.269,27.302,155.116
C02423=1059.385,-63.448,-64.953,171.271,27.303,155.116
C02424=1059.391,-63.199,-64.965,171.273,27.305,155.116
C02425=1059.398,-62.950,-64.977,171.274,27.307,155.116
C02426=1059.403,-62.699,-64.989,171.276,27.308,155.117
C02427=1059.409,-62.450,-65.000,171.279,27.310,155.117
C02428=1059.416,-62.201,-65.012,171.280,27.312,155.117
C02429=1059.422,-61.951,-65.025,171.282,27.314,155.117
C02430=1059.427,-61.701,-65.036,171.284,27.315,155.117
C02431=1059.434,-61.452,-65.048,171.285,27.317,155.117
C02432=1059.440,-61.202,-65.060,171.287,27.319,155.117
C02433=1059.446,-60.952,-65.071,171.289,27.321,155.118
C02434=1059.452,-60.703,-65.083,171.290,27.322,155.118
C02435=1059.458,-60.453,-65.096,171.292,27.324,155.118
C02436=1059.465,-60.203,-65.108,171.294,27.326,155.118
C02437=1059.472,-59.954,-65.119,171.296,27.327,155.118
C02438=1059.477,-59.704,-65.131,171.297,27.329,155.118
C02439=1059.483,-59.454,-65.143,171.299,27.331,155.118
C02440=1059.490,-59.205,-65.155,171.301,27.332,155.119
C02441=1059.496,-58.955,-65.167,171.302,27.334,155.119
C02442=1059.502,-58.706,-65.178,171.304,27.336,155.119
C02443=1059.508,-58.456,-65.190,171.306,27.338,155.119
C02444=1059.514,-58.206,-65.203,171.307,27.339,155.119
C02445=1059.521,-57.957,-65.215,171.309,27.341,155.119
C02446=1059.527,-57.708,-65.226,171.311,27.343,155.119
C02447=1059.533,-57.458,-65.239,171.312,27.344,155.120
C02448=1059.539,-57.208,-65.251,171.314,27.346,155.120
C02449=1059.545,-56.958,-65.263,171.316,27.348,155.120
C02450=1059.552,-56.708,-65.275,171.317,27.349,155.120
C02451=1059.558,-56.459,-65.286,171.319,27.351,155.120
C02452=1059.564,-56.209,-65.299,171.322,27.353,155.120
C02453=1059.570,-55.960,-65.311,171.323,27.355,155.120
C02454=1059.577,-55.710,-65.323,171.325,27.356,155.121
C02455=1059.583,-55.460,-65.335,171.327,27.358,155.121
C02456=1059.589,-55.211,-65.347,171.329,27.360,155.121
C02457=1059.595,-54.962,-65.359,171.330,27.362,155.121
C02458=1059.601,-54.711,-65.371,171.332,27.363,155.121
C02459=1059.608,-54.462,-65.383,171.334,27.365,155.121
C02460=1059.614,-54.212,-65.395,171.335,27.367,155.121
C02461=1059.620,-53.962,-65.407,171.337,27.368,155.122
C02462=1059.626,-53.712,-65.420,171.339,27.370,155.122
C02463=1059.633,-53.463,-65.432,171.340,27.372,155.122
C02464=1059.639,-53.214,-65.443,171.342,27.374,155.122
C02465=1059.645,-52.964,-65.456,171.344,27.376,155.122
C02466=1059.651,-52.715,-65.468,171.345,27.377,155.122
C02467=1059.657,-52.465,-65.480,171.347,27.379,155.123
C02468=1059.664,-52.215,-65.492,171.349,27.381,155.123
C02469=1059.671,-51.966,-65.504,171.350,27.383,155.123
C02470=1059.677,-51.716,-65.517,171.352,27.384,155.123
C02471=1059.683,-51.466,-65.529,171.354,27.386,155.123
C02472=1059.689,-51.216,-65.541,171.356,27.388,155.123
C02473=1059.696,-50.967,-65.553,171.357,27.390,155.124
C02474=1059.703,-50.688,-65.567,171.359,27.392,155.124
C02475=1059.710,-50.409,-65.581,171.361,27.394,155.124
C02476=1059.716,-50.130,-65.595,171.363,27.396,155.124
C02477=1059.723,-49.851,-65.609,171.365,27.398,155.124
C02478=1059.729,-49.601,-65.621,171.366,27.400,155.125
C02479=1059.735,-49.351,-65.634,171.368,27.401,155.125
C02480=1059.742,-49.101,-65.646,171.370,27.403,155.125
C02481=1059.748,-48.852,-65.658,171.371,27.405,155.125
C02482=1059.753,-48.602,-65.671,171.373,27.407,155.125
C02483=1059.760,-48.353,-65.683,171.375,27.409,155.125
C02484=1059.765,-48.103,-65.695,171.376,27.411,155.126
C02485=1059.772,-47.854,-65.708,171.378,27.413,155.126
C02486=1059.778,-47.604,-65.721,171.380,27.415,155.126
C02487=1059.784,-47.354,-65.733,171.381,27.417,155.126
C02488=1059.790,-47.104,-65.745,171.383,27.419,155.126
C02489=1059.796,-46.854,-65.758,171.385,27.421,155.127
C02490=1059.802,-46.605,-65.771,171.386,27.422,155.127
C02491=1059.809,-46.356,-65.783,171.388,27.424,155.127
C02492=1059.815,-46.106,-65.796,171.390,27.426,155.127
C02493=1059.820,-45.857,-65.808,171.391,27.428,155.127
C02494=1059.826,-45.607,-65.821,171.393,27.430,155.128
C02495=1059.833,-45.358,-65.833,171.394,27.432,155.128
C02496=1059.839,-45.108,-65.846,171.396,27.434,155.128
C02497=1059.845,-44.858,-65.858,171.398,27.436,155.128
C02498=1059.851,-44.608,-65.871,171.399,27.438,155.128
C02499=1059.858,-44.359,-65.884,171.401,27.439,155.128
C02500=1059.864,-44.109,-65.896,171.403,27.442,155.129
C02501=1059.869,-43.859,-65.909,171.404,27.443,155.129
C02502=1059.876,-43.610,-65.922,171.406,27.446,155.129
C02503=1059.882,-43.361,-65.934,171.409,27.448,155.129
C02504=1059.888,-43.111,-65.946,171.410,27.449,155.129
C02505=1059.894,-42.861,-65.960,171.412,27.452,155.130
C02506=1059.900,-42.612,-65.972,171.414,27.453,155.130
C02507=1059.906,-42.362,-65.985,171.415,27.456,155.130
C02508=1059.913,-42.113,-65.997,171.417,27.457,155.130
C02509=1059.919,-41.863,-66.010,171.419,27.460,155.130
C02510=1059.925,-41.613,-66.023,171.420,27.461,155.131
C02511=1059.931,-41.364,-66.036,171.422,27.463,155.131
C02512=1059.937,-41.114,-66.048,171.424,27.465,155.131
C02513=1059.944,-40.864,-66.060,171.425,27.467,155.131
C02514=1059.950,-40.615,-66.074,171.427,27.469,155.131
C02515=1059.956,-40.365,-66.086,171.429,27.471,155.132
C02516=1059.962,-40.116,-66.099,171.430,27.473,155.132
C02517=1059.968,-39.866,-66.112,171.432,27.475,155.132
C02518=1059.975,-39.616,-66.124,171.433,27.477,155.132
C02519=1059.981,-39.367,-66.137,171.435,27.479,155.132
C02520=1059.987,-39.117,-66.150,171.437,27.481,155.132
C02521=1059.993,-38.868,-66.163,171.438,27.483,155.133
C02522=1059.999,-38.618,-66.176,171.440,27.484,155.133
C02523=1060.005,-38.369,-66.189,171.442,27.487,155.133
C02524=1060.011,-38.119,-66.201,171.442,27.489,155.133
C02525=1060.017,-37.870,-66.215,171.444,27.490,155.134
C02526=1060.023,-37.620,-66.227,171.446,27.493,155.134
C02527=1060.029,-37.370,-66.241,171.447,27.494,155.134
C02528=1060.035,-37.121,-66.253,171.449,27.497,155.134
C02529=1060.042,-36.871,-66.266,171.451,27.499,155.135
C02530=1060.047,-36.621,-66.279,171.452,27.501,155.135
C02531=1060.054,-36.371,-66.293,171.454,27.503,155.135
C02532=1060.060,-36.122,-66.305,171.456,27.505,155.135
C02533=1060.066,-35.872,-66.318,171.457,27.507,155.135
C02534=1060.072,-35.622,-66.331,171.459,27.509,155.136
C02535=1060.078,-35.373,-66.344,171.460,27.511,155.136
C02536=1060.084,-35.123,-66.357,171.462,27.513,155.136
C02537=1060.091,-34.874,-66.370,171.464,27.515,155.136
C02538=1060.097,-34.595,-66.385,171.466,27.518,155.137
C02539=1060.105,-34.316,-66.399,171.468,27.520,155.137
C02540=1060.111,-34.038,-66.414,171.470,27.522,155.137
C02541=1060.117,-33.759,-66.428,171.471,27.524,155.137
C02542=1060.123,-33.510,-66.441,171.473,27.526,155.137
C02543=1060.130,-33.260,-66.455,171.474,27.529,155.138
C02544=1060.136,-33.010,-66.468,171.476,27.530,155.138
C02545=1060.142,-32.760,-66.481,171.478,27.533,155.138
C02546=1060.149,-32.511,-66.494,171.479,27.535,155.138
C02547=1060.154,-32.261,-66.507,171.481,27.537,155.139
C02548=1060.161,-32.012,-66.520,171.483,27.539,155.139
C02549=1060.167,-31.763,-66.533,171.484,27.541,155.139
C02550=1060.173,-31.513,-66.546,171.486,27.543,155.139
C02551=1060.180,-31.263,-66.559,171.487,27.545,155.140
C02552=1060.186,-31.014,-66.573,171.489,27.547,155.140
C02553=1060.191,-30.763,-66.586,171.491,27.549,155.140
C02554=1060.197,-30.514,-66.599,171.492,27.551,155.140
C02555=1060.203,-30.265,-66.612,171.494,27.554,155.140
C02556=1060.209,-30.015,-66.625,171.496,27.555,155.141
C02557=1060.216,-29.766,-66.638,171.497,27.558,155.141
C02558=1060.222,-29.516,-66.652,171.499,27.560,155.141
C02559=1060.229,-29.267,-66.665,171.501,27.562,155.141
C02560=1060.235,-29.017,-66.678,171.502,27.564,155.142
C02561=1060.241,-28.767,-66.691,171.504,27.566,155.142
C02562=1060.247,-28.518,-66.704,171.505,27.568,155.142
C02563=1060.253,-28.268,-66.718,171.507,27.570,155.142
C02564=1060.259,-28.019,-66.732,171.509,27.572,155.142
C02565=1060.265,-27.769,-66.744,171.510,27.575,155.143
C02566=1060.271,-27.519,-66.758,171.512,27.576,155.143
C02567=1060.278,-27.270,-66.771,171.513,27.578,155.143
C02568=1060.284,-27.020,-66.784,171.514,27.581,155.143
C02569=1060.291,-26.771,-66.798,171.516,27.582,155.144
C02570=1060.296,-26.521,-66.812,171.518,27.585,155.144
C02571=1060.302,-26.272,-66.824,171.519,27.587,155.144
C02572=1060.308,-26.022,-66.837,171.521,27.589,155.144
C02573=1060.314,-25.772,-66.852,171.522,27.591,155.145
C02574=1060.320,-25.523,-66.865,171.524,27.594,155.145
C02575=1060.327,-25.273,-66.878,171.526,27.596,155.145
C02576=1060.332,-25.024,-66.892,171.527,27.598,155.145
C02577=1060.338,-24.775,-66.905,171.529,27.600,155.146
C02578=1060.345,-24.525,-66.919,171.531,27.602,155.146
C02579=1060.351,-24.275,-66.933,171.532,27.604,155.146
C02580=1060.357,-24.025,-66.945,171.534,27.607,155.146
C02581=1060.363,-23.776,-66.959,171.535,27.609,155.147
C02582=1060.368,-23.526,-66.972,171.537,27.611,155.147
C02583=1060.375,-23.276,-66.986,171.539,27.613,155.147
C02584=1060.381,-23.027,-66.999,171.540,27.615,155.147
C02585=1060.387,-22.778,-67.013,171.542,27.617,155.148
C02586=1060.393,-22.528,-67.027,171.543,27.620,155.148
C02587=1060.400,-22.278,-67.040,171.545,27.622,155.148
C02588=1060.405,-22.029,-67.054,171.547,27.624,155.148
C02589=1060.412,-21.779,-67.067,171.548,27.626,155.149
C02590=1060.418,-21.530,-67.081,171.549,27.628,155.149
C02591=1060.424,-21.280,-67.095,171.551,27.631,155.149
C02592=1060.430,-21.031,-67.108,171.552,27.632,155.149
C02593=1060.436,-20.781,-67.121,171.554,27.635,155.150
C02594=1060.442,-20.531,-67.136,171.556,27.637,155.150
C02595=1060.449,-20.282,-67.149,171.557,27.639,155.150
C02596=1060.454,-20.032,-67.163,171.559,27.641,155.151
C02597=1060.460,-19.783,-67.176,171.560,27.644,155.151
C02598=1060.467,-19.534,-67.190,171.562,27.646,155.151
C02599=1060.473,-19.284,-67.204,171.564,27.648,155.151
C02600=1060.479,-19.035,-67.217,171.565,27.651,155.152
C02601=1060.486,-18.785,-67.231,171.567,27.653,155.152
C02602=1060.492,-18.505,-67.246,171.568,27.655,155.152
C02603=1060.499,-18.226,-67.262,171.570,27.657,155.152
C02604=1060.506,-17.946,-67.277,171.572,27.660,155.153
C02605=1060.513,-17.666,-67.292,171.574,27.663,155.153
C02606=1060.519,-17.417,-67.306,171.576,27.664,155.153
C02607=1060.525,-17.168,-67.320,171.577,27.667,155.153
C02608=1060.531,-16.918,-67.334,171.578,27.669,155.154
C02609=1060.538,-16.668,-67.347,171.580,27.671,155.154
C02610=1060.543,-16.419,-67.361,171.581,27.673,155.154
C02611=1060.550,-16.169,-67.375,171.583,27.675,155.155
C02612=1060.556,-15.920,-67.389,171.585,27.678,155.155
C02613=1060.563,-15.670,-67.403,171.586,27.680,155.155
C02614=1060.569,-15.421,-67.416,171.588,27.682,155.155
C02615=1060.574,-15.171,-67.430,171.589,27.684,155.156
C02616=1060.581,-14.921,-67.444,171.591,27.687,155.156
C02617=1060.587,-14.672,-67.458,171.593,27.689,155.156
C02618=1060.592,-14.423,-67.472,171.594,27.691,155.156
C02619=1060.599,-14.173,-67.486,171.596,27.694,155.157
C02620=1060.605,-13.923,-67.500,171.597,27.696,155.157
C02621=1060.610,-13.674,-67.514,171.599,27.698,155.157
C02622=1060.617,-13.424,-67.528,171.601,27.700,155.157
C02623=1060.623,-13.175,-67.542,171.601,27.702,155.158
C02624=1060.629,-12.925,-67.555,171.603,27.705,155.158
C02625=1060.635,-12.676,-67.570,171.605,27.707,155.158
C02626=1060.641,-12.426,-67.584,171.606,27.710,155.159
C02627=1060.648,-12.176,-67.597,171.608,27.712,155.159
C02628=1060.653,-11.927,-67.612,171.609,27.714,155.159
C02629=1060.659,-11.678,-67.626,171.611,27.716,155.159
C02630=1060.666,-11.428,-67.639,171.613,27.719,155.160
C02631=1060.671,-11.179,-67.654,171.614,27.721,155.160
C02632=1060.678,-10.928,-67.668,171.616,27.723,155.160
C02633=1060.684,-10.679,-67.682,171.617,27.725,155.161
C02634=1060.690,-10.430,-67.696,171.619,27.728,155.161
C02635=1060.696,-10.180,-67.710,171.621,27.730,155.161
C02636=1060.702,-9.931,-67.724,171.621,27.732,155.161
C02637=1060.708,-9.681,-67.739,171.623,27.734,155.162
C02638=1060.714,-9.432,-67.752,171.624,27.737,155.162
C02639=1060.721,-9.182,-67.767,171.626,27.739,155.162
C02640=1060.726,-8.933,-67.781,171.628,27.742,155.163
C02641=1060.732,-8.683,-67.794,171.629,27.744,155.163
C02642=1060.739,-8.434,-67.809,171.631,27.746,155.163
C02643=1060.744,-8.184,-67.823,171.633,27.748,155.163
C02644=1060.751,-7.934,-67.838,171.634,27.751,155.164
C02645=1060.757,-7.685,-67.851,171.636,27.753,155.164
C02646=1060.763,-7.435,-67.866,171.637,27.755,155.164
C02647=1060.769,-7.186,-67.880,171.639,27.757,155.164
C02648=1060.776,-6.937,-67.894,171.641,27.760,155.165
C02649=1060.781,-6.687,-67.908,171.641,27.762,155.165
C02650=1060.788,-6.437,-67.923,171.643,27.765,155.165
C02651=1060.794,-6.188,-67.936,171.644,27.767,155.166
C02652=1060.800,-5.938,-67.950,171.646,27.769,155.166
C02653=1060.806,-5.689,-67.965,171.648,27.771,155.166
C02654=1060.813,-5.439,-67.979,171.649,27.774,155.167
C02655=1060.818,-5.190,-67.993,171.651,27.776,155.167
C02656=1060.825,-4.940,-68.008,171.653,27.778,155.167
C02657=1060.830,-4.691,-68.022,171.654,27.781,155.167
C02658=1060.837,-4.441,-68.036,171.656,27.783,155.168
C02659=1060.843,-4.192,-68.050,171.657,27.785,155.168
C02660=1060.849,-3.942,-68.065,171.658,27.787,155.168
C02661=1060.855,-3.693,-68.078,171.660,27.790,155.169
C02662=1060.862,-3.443,-68.093,171.661,27.792,155.169
C02663=1060.868,-3.194,-68.108,171.663,27.794,155.169
C02664=1060.874,-2.944,-68.122,171.664,27.797,155.169
C02665=1060.880,-2.695,-68.137,171.666,27.799,155.170
C02666=1060.887,-2.413,-68.153,171.668,27.802,155.170
C02667=1060.893,-2.132,-68.169,171.669,27.804,155.170
C02668=1060.900,-1.851,-68.186,171.671,27.807,155.171
C02669=1060.907,-1.570,-68.202,171.673,27.810,155.171
C02670=1060.913,-1.320,-68.217,171.674,27.812,155.171
C02671=1060.919,-1.071,-68.231,171.675,27.815,155.172
C02672=1060.925,-0.821,-68.246,171.677,27.817,155.172
C02673=1060.931,-0.572,-68.260,171.679,27.820,155.172
C02674=1060.937,-0.322,-68.275,171.680,27.822,155.173
C02675=1060.943,-0.073,-68.289,171.682,27.825,155.173
C02676=1060.949,0.177,-68.304,171.683,27.827,155.173
C02677=1060.955,0.426,-68.319,171.685,27.829,155.174
C02678=1060.961,0.676,-68.333,171.687,27.832,155.174
C02679=1060.967,0.925,-68.348,171.688,27.834,155.174
C02680=1060.973,1.175,-68.362,171.689,27.836,155.175
C02681=1060.978,1.424,-68.376,171.690,27.839,155.175
C02682=1060.985,1.674,-68.391,171.692,27.841,155.175
C02683=1060.991,1.923,-68.406,171.694,27.844,155.175
C02684=1060.997,2.173,-68.421,171.695,27.846,155.176
C02685=1061.003,2.422,-68.436,171.697,27.849,155.176
C02686=1061.009,2.672,-68.450,171.698,27.851,155.176
C02687=1061.015,2.922,-68.465,171.700,27.853,155.177
C02688=1061.021,3.170,-68.479,171.702,27.856,155.177
C02689=1061.027,3.420,-68.494,171.702,27.858,155.177
C02690=1061.034,3.670,-68.509,171.704,27.860,155.178
C02691=1061.039,3.919,-68.523,171.705,27.863,155.178
C02692=1061.046,4.169,-68.538,171.707,27.865,155.178
C02693=1061.051,4.418,-68.552,171.709,27.868,155.179
C02694=1061.058,4.668,-68.567,171.710,27.870,155.179
C02695=1061.064,4.917,-68.582,171.712,27.873,155.179
C02696=1061.070,5.166,-68.597,171.713,27.875,155.179
C02697=1061.075,5.417,-68.612,171.715,27.877,155.180
C02698=1061.081,5.666,-68.626,171.716,27.880,155.180
C02699=1061.087,5.915,-68.641,171.717,27.882,155.180
C02700=1061.094,6.165,-68.656,171.719,27.884,155.181
C02701=1061.100,6.414,-68.671,171.720,27.887,155.181
C02702=1061.106,6.664,-68.686,171.722,27.889,155.181
C02703=1061.112,6.913,-68.701,171.724,27.892,155.182
C02704=1061.118,7.162,-68.715,171.725,27.894,155.182
C02705=1061.125,7.412,-68.730,171.727,27.897,155.182
C02706=1061.131,7.662,-68.745,171.728,27.899,155.183
C02707=1061.137,7.911,-68.760,171.729,27.902,155.183
C02708=1061.143,8.160,-68.775,171.731,27.904,155.183
C02709=1061.149,8.411,-68.789,171.732,27.906,155.184
C02710=1061.155,8.659,-68.803,171.734,27.909,155.184
C02711=1061.161,8.909,-68.819,171.736,27.911,155.184
C02712=1061.167,9.159,-68.834,171.737,27.913,155.184
C02713=1061.173,9.409,-68.849,171.739,27.916,155.185
C02714=1061.179,9.658,-68.863,171.740,27.918,155.185
C02715=1061.186,9.907,-68.878,171.741,27.920,155.185
C02716=1061.192,10.157,-68.893,171.743,27.923,155.186
C02717=1061.198,10.406,-68.908,171.744,27.925,155.186
C02718=1061.204,10.656,-68.923,171.746,27.928,155.186
C02719=1061.211,10.905,-68.939,171.747,27.931,155.187
C02720=1061.217,11.154,-68.954,171.749,27.933,155.187
C02721=1061.222,11.404,-68.969,171.751,27.935,155.187
C02722=1061.229,11.653,-68.984,171.752,27.938,155.188
C02723=1061.235,11.903,-68.999,171.753,27.940,155.188
C02724=1061.241,12.153,-69.014,171.754,27.942,155.188
C02725=1061.247,12.402,-69.028,171.756,27.945,155.189
C02726=1061.254,12.651,-69.043,171.758,27.947,155.189
C02727=1061.260,12.901,-69.058,171.759,27.949,155.189
C02728=1061.266,13.150,-69.073,171.761,27.952,155.190
C02729=1061.272,13.399,-69.088,171.762,27.954,155.190
C02730=1061.279,13.683,-69.105,171.764,27.957,155.190
C02731=1061.286,13.965,-69.122,171.766,27.960,155.191
C02732=1061.292,14.249,-69.139,171.767,27.962,155.191
C02733=1061.300,14.532,-69.156,171.769,27.965,155.191
C02734=1061.306,14.782,-69.171,171.770,27.968,155.192
C02735=1061.312,15.031,-69.187,171.772,27.970,155.192
C02736=1061.319,15.281,-69.202,171.773,27.973,155.192
C02737=1061.324,15.530,-69.217,171.775,27.975,155.193
C02738=1061.330,15.780,-69.233,171.777,27.978,155.193
C02739=1061.336,16.029,-69.247,171.777,27.980,155.193
C02740=1061.343,16.278,-69.263,171.779,27.982,155.194
C02741=1061.348,16.528,-69.278,171.781,27.985,155.194
C02742=1061.354,16.777,-69.293,171.782,27.987,155.194
C02743=1061.361,17.027,-69.308,171.784,27.990,155.195
C02744=1061.367,17.276,-69.324,171.785,27.993,155.195
C02745=1061.373,17.526,-69.339,171.787,27.995,155.195
C02746=1061.378,17.775,-69.355,171.788,27.997,155.196
C02747=1061.385,18.025,-69.370,171.789,28.000,155.196
C02748=1061.391,18.274,-69.385,171.791,28.002,155.196
C02749=1061.397,18.524,-69.401,171.792,28.005,155.197
C02750=1061.403,18.774,-69.416,171.794,28.007,155.197
C02751=1061.409,19.022,-69.431,171.795,28.010,155.197
C02752=1061.415,19.272,-69.447,171.797,28.012,155.198
C02753=1061.421,19.522,-69.461,171.799,28.015,155.198
C02754=1061.427,19.771,-69.477,171.799,28.017,155.198
C02755=1061.434,20.021,-69.493,171.801,28.020,155.199
C02756=1061.440,20.270,-69.508,171.803,28.022,155.199
C02757=1061.445,20.519,-69.524,171.804,28.025,155.199
C02758=1061.452,20.768,-69.538,171.806,28.027,155.200
C02759=1061.458,21.018,-69.554,171.807,28.030,155.200
C02760=1061.464,21.267,-69.570,171.809,28.032,155.200
C02761=1061.470,21.517,-69.585,171.810,28.035,155.201
C02762=1061.476,21.767,-69.600,171.811,28.037,155.201
C02763=1061.482,22.016,-69.616,171.813,28.040,155.201
C02764=1061.488,22.265,-69.631,171.814,28.042,155.202
C02765=1061.494,22.515,-69.647,171.816,28.045,155.202
C02766=1061.500,22.764,-69.662,171.818,28.047,155.202
C02767=1061.506,23.014,-69.678,171.819,28.050,155.203
C02768=1061.513,23.263,-69.693,171.820,28.052,155.203
C02769=1061.518,23.513,-69.709,171.821,28.055,155.203
C02770=1061.524,23.762,-69.724,171.823,28.057,155.204
C02771=1061.530,24.012,-69.740,171.825,28.060,155.204
C02772=1061.537,24.261,-69.755,171.826,28.062,155.204
C02773=1061.542,24.511,-69.771,171.828,28.065,155.205
C02774=1061.549,24.760,-69.787,171.829,28.068,155.205
C02775=1061.555,25.010,-69.802,171.830,28.070,155.205
C02776=1061.561,25.259,-69.818,171.832,28.073,155.206
C02777=1061.567,25.509,-69.833,171.833,28.075,155.206
C02778=1061.572,25.757,-69.849,171.835,28.078,155.206
C02779=1061.579,26.007,-69.864,171.836,28.080,155.207
C02780=1061.585,26.256,-69.880,171.838,28.083,155.207
C02781=1061.591,26.506,-69.895,171.839,28.085,155.207
C02782=1061.597,26.755,-69.912,171.840,28.088,155.208
C02783=1061.604,27.004,-69.927,171.842,28.090,155.208
C02784=1061.609,27.254,-69.943,171.843,28.093,155.208
C02785=1061.615,27.504,-69.959,171.845,28.095,155.209
C02786=1061.622,27.753,-69.974,171.847,28.098,155.209
C02787=1061.628,28.003,-69.990,171.848,28.101,155.210
C02788=1061.634,28.252,-70.005,171.849,28.103,155.210
C02789=1061.640,28.502,-70.022,171.850,28.105,155.210
C02790=1061.646,28.751,-70.038,171.852,28.108,155.211
C02791=1061.652,29.001,-70.053,171.854,28.110,155.211
C02792=1061.658,29.249,-70.069,171.855,28.113,155.211
C02793=1061.664,29.499,-70.085,171.857,28.115,155.212
C02794=1061.671,29.784,-70.103,171.858,28.118,155.212
C02795=1061.678,30.068,-70.121,171.860,28.121,155.212
C02796=1061.685,30.353,-70.138,171.861,28.124,155.213
C02797=1061.691,30.637,-70.157,171.863,28.127,155.213
C02798=1061.697,30.886,-70.172,171.865,28.129,155.214
C02799=1061.703,31.136,-70.188,171.866,28.132,155.214
C02800=1061.709,31.385,-70.205,171.868,28.135,155.214
C02801=1061.715,31.635,-70.221,171.868,28.137,155.215
C02802=1061.722,31.884,-70.236,171.870,28.140,155.215
C02803=1061.728,32.134,-70.252,171.872,28.142,155.215
C02804=1061.734,32.383,-70.268,171.873,28.145,155.216
C02805=1061.739,32.633,-70.284,171.875,28.148,155.216
C02806=1061.745,32.882,-70.300,171.876,28.150,155.216
C02807=1061.752,33.131,-70.316,171.878,28.153,155.217
C02808=1061.758,33.381,-70.332,171.879,28.155,155.217
C02809=1061.764,33.631,-70.348,171.880,28.158,155.217
C02810=1061.769,33.880,-70.364,171.882,28.160,155.218
C02811=1061.776,34.129,-70.379,171.883,28.163,155.218
C02812=1061.782,34.378,-70.396,171.885,28.165,155.219
C02813=1061.788,34.628,-70.412,171.887,28.168,155.219
C02814=1061.794,34.878,-70.428,171.887,28.170,155.219
C02815=1061.800,35.127,-70.443,171.889,28.173,155.220
C02816=1061.806,35.376,-70.459,171.890,28.175,155.220
C02817=1061.812,35.625,-70.476,171.892,28.178,155.220
C02818=1061.818,35.875,-70.492,171.894,28.181,155.221
C02819=1061.824,36.124,-70.508,171.895,28.183,155.221
C02820=1061.831,36.373,-70.524,171.897,28.186,155.221
C02821=1061.837,36.623,-70.539,171.897,28.188,155.222
C02822=1061.842,36.872,-70.556,171.899,28.191,155.222
C02823=1061.848,37.122,-70.572,171.901,28.194,155.222
C02824=1061.854,37.371,-70.588,171.902,28.196,155.223
C02825=1061.862,37.621,-70.604,171.904,28.199,155.223
C02826=1061.868,37.870,-70.620,171.905,28.201,155.223
C02827=1061.874,38.120,-70.637,171.906,28.203,155.224
C02828=1061.880,38.369,-70.653,171.908,28.206,155.224
C02829=1061.885,38.618,-70.669,171.909,28.209,155.225
C02830=1061.891,38.868,-70.685,171.911,28.211,155.225
C02831=1061.897,39.117,-70.702,171.912,28.214,155.225
C02832=1061.903,39.366,-70.718,171.914,28.217,155.226
C02833=1061.909,39.616,-70.734,171.915,28.219,155.226
C02834=1061.915,39.866,-70.750,171.916,28.222,155.226
C02835=1061.921,40.115,-70.766,171.918,28.224,155.227
C02836=1061.927,40.364,-70.782,171.919,28.227,155.227
C02837=1061.933,40.614,-70.799,171.921,28.229,155.227
C02838=1061.939,40.863,-70.815,171.923,28.232,155.228
C02839=1061.945,41.112,-70.831,171.923,28.235,155.228
C02840=1061.951,41.361,-70.848,171.925,28.238,155.229
C02841=1061.957,41.610,-70.864,171.926,28.240,155.229
C02842=1061.963,41.860,-70.881,171.928,28.243,155.229
C02843=1061.969,42.110,-70.897,171.930,28.245,155.230
C02844=1061.975,42.359,-70.913,171.931,28.248,155.230
C02845=1061.981,42.609,-70.930,171.933,28.250,155.230
C02846=1061.987,42.858,-70.946,171.933,28.253,155.231
C02847=1061.993,43.107,-70.962,171.935,28.255,155.231
C02848=1061.999,43.357,-70.978,171.937,28.258,155.231
C02849=1062.005,43.606,-70.995,171.938,28.261,155.232
C02850=1062.010,43.856,-71.012,171.940,28.264,155.232
C02851=1062.017,44.106,-71.028,171.941,28.266,155.233
C02852=1062.023,44.355,-71.044,171.942,28.268,155.233
C02853=1062.029,44.604,-71.061,171.944,28.271,155.233
C02854=1062.035,44.853,-71.078,171.945,28.274,155.234
C02855=1062.040,45.103,-71.095,171.947,28.277,155.234
C02856=1062.046,45.352,-71.111,171.948,28.279,155.234
C02857=1062.052,45.601,-71.127,171.950,28.282,155.235
C02858=1062.059,45.886,-71.146,171.952,28.285,155.235
C02859=1062.066,46.170,-71.165,171.953,28.288,155.236
C02860=1062.073,46.454,-71.184,171.955,28.291,155.236
C02861=1062.080,46.739,-71.203,171.956,28.294,155.237
C02862=1062.085,46.989,-71.220,171.958,28.297,155.237
C02863=1062.091,47.238,-71.236,171.959,28.299,155.237
C02864=1062.097,47.487,-71.252,171.960,28.302,155.238
C02865=1062.102,47.736,-71.270,171.962,28.305,155.238
C02866=1062.108,47.986,-71.286,171.963,28.307,155.238
C02867=1062.115,48.236,-71.303,171.965,28.310,155.239
C02868=1062.121,48.485,-71.319,171.966,28.312,155.239
C02869=1062.126,48.734,-71.337,171.968,28.315,155.240
C02870=1062.132,48.983,-71.353,171.969,28.318,155.240
C02871=1062.138,49.233,-71.369,171.970,28.320,155.240
C02872=1062.144,49.482,-71.386,171.972,28.323,155.241
C02873=1062.150,49.732,-71.403,171.973,28.325,155.241
C02874=1062.156,49.981,-71.420,171.975,28.328,155.241
C02875=1062.162,50.230,-71.437,171.977,28.331,155.242
C02876=1062.168,50.479,-71.453,171.977,28.334,155.242
C02877=1062.174,50.729,-71.470,171.979,28.336,155.243
C02878=1062.180,50.978,-71.487,171.980,28.339,155.243
C02879=1062.186,51.228,-71.503,171.982,28.341,155.243
C02880=1062.192,51.477,-71.520,171.984,28.344,155.244
C02881=1062.198,51.726,-71.537,171.985,28.347,155.244
C02882=1062.204,51.976,-71.553,171.986,28.349,155.244
C02883=1062.210,52.226,-71.571,171.987,28.352,155.245
C02884=1062.216,52.475,-71.588,171.989,28.355,155.245
C02885=1062.222,52.724,-71.604,171.991,28.357,155.246
C02886=1062.228,52.973,-71.621,171.992,28.360,155.246
C02887=1062.233,53.222,-71.638,171.994,28.362,155.246
C02888=1062.240,53.472,-71.654,171.995,28.365,155.247
C02889=1062.246,53.721,-71.671,171.996,28.368,155.247
C02890=1062.251,53.971,-71.688,171.998,28.371,155.247
C02891=1062.258,54.220,-71.705,171.999,28.373,155.248
C02892=1062.264,54.470,-71.722,172.001,28.376,155.248
C02893=1062.270,54.719,-71.739,172.002,28.378,155.249
C02894=1062.276,54.968,-71.755,172.003,28.381,155.249
C02895=1062.282,55.217,-71.773,172.005,28.383,155.249
C02896=1062.288,55.467,-71.790,172.006,28.386,155.250
C02897=1062.294,55.716,-71.807,172.008,28.389,155.250
C02898=1062.300,55.965,-71.823,172.010,28.391,155.250
C02899=1062.306,56.215,-71.841,172.011,28.394,155.251
C02900=1062.312,56.464,-71.857,172.012,28.396,155.251
C02901=1062.318,56.713,-71.874,172.013,28.399,155.252
C02902=1062.324,56.963,-71.891,172.015,28.402,155.252
C02903=1062.330,57.212,-71.908,172.017,28.405,155.252
C02904=1062.336,57.461,-71.924,172.018,28.407,155.253
C02905=1062.342,57.711,-71.942,172.020,28.410,155.253
C02906=1062.348,57.960,-71.959,172.020,28.412,155.253
C02907=1062.354,58.210,-71.976,172.022,28.415,155.254
C02908=1062.360,58.460,-71.993,172.024,28.417,155.254
C02909=1062.367,58.708,-72.010,172.025,28.420,155.255
C02910=1062.372,58.957,-72.027,172.027,28.423,155.255
C02911=1062.379,59.207,-72.044,172.029,28.425,155.255
C02912=1062.385,59.456,-72.061,172.029,28.427,155.256
C02913=1062.390,59.706,-72.078,172.031,28.430,155.256
C02914=1062.397,59.955,-72.095,172.032,28.433,155.256
C02915=1062.403,60.204,-72.112,172.034,28.435,155.257
C02916=1062.409,60.454,-72.129,172.036,28.438,155.257
C02917=1062.415,60.703,-72.146,172.037,28.441,155.257
C02918=1062.421,60.952,-72.164,172.039,28.444,155.258
C02919=1062.427,61.202,-72.181,172.040,28.446,155.258
C02920=1062.434,61.451,-72.198,172.041,28.448,155.259
C02921=1062.440,61.701,-72.215,172.043,28.451,155.259
C02922=1062.446,61.985,-72.234,172.044,28.454,155.259
C02923=1062.454,62.269,-72.254,172.046,28.457,155.260
C02924=1062.461,62.553,-72.273,172.047,28.460,155.260
C02925=1062.467,62.837,-72.293,172.049,28.463,155.261
C02926=1062.474,63.086,-72.310,172.051,28.465,155.261
C02927=1062.480,63.336,-72.327,172.052,28.468,155.261
C02928=1062.486,63.585,-72.345,172.054,28.471,155.262
C02929=1062.492,63.834,-72.362,172.055,28.473,155.262
C02930=1062.498,64.083,-72.379,172.057,28.476,155.262
C02931=1062.505,64.334,-72.396,172.059,28.478,155.263
C02932=1062.510,64.583,-72.414,172.059,28.481,155.263
C02933=1062.516,64.831,-72.431,172.061,28.484,155.264
C02934=1062.522,65.081,-72.449,172.062,28.487,155.264
C02935=1062.528,65.331,-72.465,172.064,28.489,155.264
C02936=1062.534,65.580,-72.483,172.066,28.492,155.265
C02937=1062.540,65.829,-72.500,172.067,28.494,155.265
C02938=1062.546,66.078,-72.518,172.068,28.497,155.266
C02939=1062.552,66.328,-72.535,172.070,28.500,155.266
C02940=1062.558,66.577,-72.553,172.071,28.502,155.266
C02941=1062.564,66.827,-72.569,172.073,28.505,155.267
C02942=1062.570,67.076,-72.587,172.074,28.507,155.267
C02943=1062.576,67.326,-72.605,172.076,28.510,155.267
C02944=1062.582,67.574,-72.622,172.078,28.513,155.268
C02945=1062.588,67.824,-72.640,172.078,28.516,155.268
C02946=1062.594,68.073,-72.657,172.080,28.518,155.269
C02947=1062.599,68.322,-72.675,172.082,28.520,155.269
C02948=1062.606,68.572,-72.692,172.083,28.523,155.269
C02949=1062.612,68.821,-72.710,172.085,28.526,155.270
C02950=1062.618,69.070,-72.728,172.086,28.529,155.270
C02951=1062.624,69.320,-72.744,172.087,28.531,155.271
C02952=1062.630,69.569,-72.762,172.089,28.534,155.271
C02953=1062.636,69.818,-72.780,172.090,28.536,155.271
C02954=1062.642,70.068,-72.798,172.092,28.539,155.272
C02955=1062.648,70.317,-72.814,172.093,28.542,155.272
C02956=1062.654,70.567,-72.832,172.095,28.545,155.272
C02957=1062.660,70.816,-72.850,172.096,28.547,155.273
C02958=1062.665,71.065,-72.868,172.097,28.550,155.273
C02959=1062.671,71.314,-72.885,172.099,28.553,155.274
C02960=1062.677,71.563,-72.902,172.101,28.555,155.274
C02961=1062.684,71.813,-72.920,172.102,28.558,155.274
C02962=1062.689,72.062,-72.938,172.104,28.561,155.275
C02963=1062.695,72.312,-72.956,172.105,28.563,155.275
C02964=1062.701,72.561,-72.973,172.106,28.566,155.276
C02965=1062.707,72.810,-72.991,172.108,28.569,155.276
C02966=1062.713,73.059,-73.009,172.109,28.571,155.276
C02967=1062.720,73.308,-73.027,172.111,28.574,155.277
C02968=1062.725,73.557,-73.045,172.112,28.576,155.277
C02969=1062.731,73.807,-73.062,172.114,28.579,155.277
C02970=1062.737,74.056,-73.080,172.115,28.582,155.278
C02971=1062.743,74.306,-73.098,172.116,28.584,155.278
C02972=1062.748,74.555,-73.116,172.118,28.587,155.279
C02973=1062.755,74.804,-73.133,172.120,28.590,155.279
C02974=1062.761,75.053,-73.150,172.121,28.593,155.279
C02975=1062.767,75.303,-73.168,172.123,28.595,155.280
C02976=1062.773,75.552,-73.187,172.124,28.598,155.280
C02977=1062.779,75.801,-73.205,172.125,28.600,155.281
C02978=1062.785,76.051,-73.223,172.127,28.603,155.281
C02979=1062.790,76.300,-73.240,172.128,28.606,155.281
C02980=1062.797,76.550,-73.258,172.130,28.609,155.282
C02981=1062.802,76.799,-73.276,172.131,28.611,155.282
C02982=1062.809,77.048,-73.294,172.133,28.614,155.282
C02983=1062.815,77.297,-73.311,172.135,28.616,155.283
C02984=1062.821,77.546,-73.329,172.135,28.619,155.283
C02985=1062.827,77.796,-73.347,172.137,28.622,155.284
C02986=1062.833,78.079,-73.368,172.139,28.624,155.284
C02987=1062.840,78.364,-73.388,172.140,28.628,155.285
C02988=1062.847,78.648,-73.409,172.143,28.631,155.285
C02989=1062.853,78.932,-73.429,172.144,28.634,155.285
C02990=1062.859,79.182,-73.447,172.146,28.637,155.286
C02991=1062.866,79.431,-73.466,172.146,28.639,155.286
C02992=1062.871,79.680,-73.483,172.148,28.642,155.287
C02993=1062.877,79.930,-73.501,172.150,28.644,155.287
C02994=1062.883,80.178,-73.519,172.151,28.647,155.287
C02995=1062.889,80.428,-73.537,172.153,28.650,155.288
C02996=1062.895,80.677,-73.555,172.155,28.653,155.288
C02997=1062.901,80.926,-73.574,172.156,28.655,155.289
C02998=1062.907,81.176,-73.592,172.157,28.658,155.289
C02999=1062.912,81.425,-73.610,172.158,28.661,155.289
C03000=1062.919,81.674,-73.628,172.160,28.664,155.290
C03001=1062.924,81.923,-73.646,172.162,28.666,155.290
C03002=1062.930,82.173,-73.664,172.163,28.669,155.291
C03003=1062.936,82.421,-73.682,172.165,28.672,155.291
C03004=1062.942,82.671,-73.700,172.166,28.674,155.291
C03005=1062.949,82.920,-73.719,172.167,28.677,155.292
C03006=1062.953,83.169,-73.737,172.169,28.680,155.292
C03007=1062.959,83.419,-73.755,172.170,28.682,155.292
C03008=1062.966,83.668,-73.773,172.172,28.685,155.293
C03009=1062.971,83.917,-73.791,172.174,28.688,155.293
C03010=1062.978,84.167,-73.810,172.175,28.690,155.294
C03011=1062.984,84.416,-73.828,172.177,28.693,155.294
C03012=1062.989,84.665,-73.846,172.178,28.696,155.295
C03013=1062.995,84.915,-73.864,172.179,28.699,155.295
C03014=1063.001,85.164,-73.882,172.181,28.701,155.295
C03015=1063.007,85.413,-73.901,172.182,28.704,155.296
C03016=1063.013,85.663,-73.918,172.184,28.707,155.296
C03017=1063.019,85.911,-73.937,172.186,28.709,155.296
C03018=1063.024,86.161,-73.955,172.187,28.712,155.297
C03019=1063.031,86.410,-73.974,172.188,28.714,155.297
C03020=1063.037,86.660,-73.992,172.190,28.717,155.298
C03021=1063.043,86.908,-74.010,172.191,28.720,155.298
C03022=1063.049,87.158,-74.028,172.193,28.723,155.298
C03023=1063.055,87.407,-74.047,172.194,28.725,155.299
C03024=1063.060,87.656,-74.066,172.196,28.728,155.299
C03025=1063.067,87.906,-74.084,172.198,28.731,155.300
C03026=1063.073,88.155,-74.102,172.199,28.733,155.300
C03027=1063.078,88.404,-74.120,172.200,28.736,155.300
C03028=1063.085,88.653,-74.138,172.202,28.738,155.301
C03029=1063.090,88.903,-74.157,172.203,28.741,155.301
C03030=1063.097,89.152,-74.176,172.205,28.744,155.302
C03031=1063.103,89.401,-74.194,172.206,28.747,155.302
C03032=1063.109,89.650,-74.212,172.208,28.749,155.302
C03033=1063.115,89.899,-74.230,172.210,28.752,155.303
C03034=1063.120,90.150,-74.249,172.211,28.754,155.303
C03035=1063.126,90.398,-74.267,172.212,28.757,155.303
C03036=1063.133,90.647,-74.286,172.214,28.760,155.304
C03037=1063.139,90.897,-74.304,172.215,28.762,155.304
C03038=1063.145,91.146,-74.323,172.217,28.765,155.305
C03039=1063.150,91.395,-74.341,172.218,28.768,155.305
C03040=1063.156,91.645,-74.360,172.220,28.771,155.305
C03041=1063.162,91.894,-74.379,172.222,28.773,155.306
C03042=1063.168,92.142,-74.397,172.223,28.776,155.306
C03043=1063.174,92.392,-74.416,172.224,28.779,155.307
C03044=1063.180,92.641,-74.434,172.226,28.781,155.307
C03045=1063.185,92.891,-74.453,172.227,28.784,155.307
C03046=1063.191,93.139,-74.472,172.229,28.787,155.308
C03047=1063.197,93.389,-74.491,172.230,28.790,155.308
C03048=1063.203,93.638,-74.509,172.232,28.793,155.309
C03049=1063.209,93.888,-74.528,172.234,28.795,155.309
C03050=1063.216,94.172,-74.549,172.235,28.798,155.309
C03051=1063.223,94.456,-74.570,172.237,28.801,155.310
C03052=1063.229,94.740,-74.592,172.238,28.804,155.310
C03053=1063.236,95.024,-74.613,172.240,28.807,155.311
C03054=1063.241,95.273,-74.631,172.242,28.810,155.311
C03055=1063.247,95.522,-74.650,172.243,28.812,155.312
C03056=1063.253,95.771,-74.669,172.245,28.815,155.312
C03057=1063.260,96.020,-74.688,172.247,28.818,155.312
C03058=1063.266,96.270,-74.706,172.248,28.821,155.313
C03059=1063.271,96.519,-74.725,172.250,28.823,155.313
C03060=1063.277,96.768,-74.743,172.251,28.826,155.314
C03061=1063.283,97.017,-74.763,172.252,28.829,155.314
C03062=1063.289,97.267,-74.781,172.254,28.831,155.314
C03063=1063.295,97.516,-74.801,172.255,28.834,155.315
C03064=1063.301,97.764,-74.819,172.257,28.837,155.315
C03065=1063.307,98.014,-74.838,172.259,28.840,155.316
C03066=1063.313,98.263,-74.857,172.260,28.842,155.316
C03067=1063.318,98.513,-74.875,172.262,28.845,155.316
C03068=1063.325,98.762,-74.894,172.264,28.847,155.317
C03069=1063.330,99.012,-74.913,172.265,28.850,155.317
C03070=1063.337,99.261,-74.932,172.266,28.853,155.318
C03071=1063.342,99.509,-74.951,172.267,28.855,155.318
C03072=1063.348,99.759,-74.969,172.269,28.858,155.318
C03073=1063.354,100.008,-74.989,172.271,28.861,155.319
C03074=1063.361,100.257,-75.007,172.272,28.864,155.319
C03075=1063.366,100.507,-75.027,172.274,28.866,155.320
C03076=1063.373,100.756,-75.045,172.276,28.869,155.320
C03077=1063.378,101.005,-75.064,172.277,28.871,155.320
C03078=1063.384,101.255,-75.084,172.279,28.874,155.321
C03079=1063.390,101.503,-75.102,172.281,28.877,155.321
C03080=1063.396,101.752,-75.121,172.281,28.879,155.322
C03081=1063.401,102.002,-75.140,172.283,28.882,155.322
C03082=1063.407,102.251,-75.160,172.285,28.885,155.322
C03083=1063.413,102.500,-75.178,172.286,28.888,155.323
C03084=1063.419,102.750,-75.198,172.288,28.890,155.323
C03085=1063.425,102.999,-75.218,172.289,28.893,155.324
C03086=1063.431,103.247,-75.236,172.291,28.896,155.324
C03087=1063.437,103.497,-75.255,172.293,28.899,155.324
C03088=1063.442,103.746,-75.274,172.294,28.901,155.325
C03089=1063.448,103.995,-75.294,172.296,28.904,155.325
C03090=1063.454,104.245,-75.312,172.297,28.907,155.326
C03091=1063.460,104.494,-75.331,172.298,28.909,155.326
C03092=1063.466,104.743,-75.351,172.300,28.912,155.326
C03093=1063.471,104.993,-75.370,172.301,28.915,155.327
C03094=1063.478,105.241,-75.389,172.303,28.918,155.327
C03095=1063.483,105.490,-75.408,172.305,28.920,155.328
C03096=1063.489,105.739,-75.427,172.306,28.923,155.328
C03097=1063.495,105.989,-75.447,172.308,28.926,155.328
C03098=1063.501,106.238,-75.465,172.310,28.929,155.329
C03099=1063.507,106.487,-75.485,172.311,28.931,155.329
C03100=1063.513,106.736,-75.504,172.313,28.934,155.330
C03101=1063.518,106.986,-75.524,172.315,28.937,155.330
C03102=1063.525,107.235,-75.542,172.315,28.939,155.330
C03103=1063.530,107.484,-75.562,172.317,28.942,155.331
C03104=1063.536,107.733,-75.582,172.318,28.945,155.331
C03105=1063.542,107.983,-75.601,172.320,28.948,155.332
C03106=1063.548,108.232,-75.620,172.322,28.950,155.332
C03107=1063.554,108.481,-75.639,172.323,28.953,155.332
C03108=1063.560,108.730,-75.659,172.325,28.956,155.333
C03109=1063.566,108.979,-75.678,172.327,28.959,155.333
C03110=1063.572,109.229,-75.697,172.328,28.961,155.334
C03111=1063.578,109.478,-75.717,172.330,28.964,155.334
C03112=1063.584,109.727,-75.736,172.332,28.966,155.334
C03113=1063.590,109.976,-75.755,172.333,28.969,155.335
C03114=1063.596,110.260,-75.777,172.335,28.972,155.335
C03115=1063.603,110.544,-75.799,172.336,28.975,155.336
C03116=1063.610,110.828,-75.822,172.338,28.978,155.336
C03117=1063.617,111.112,-75.843,172.340,28.981,155.337
C03118=1063.623,111.335,-75.861,172.341,28.984,155.337
C03119=1063.628,111.558,-75.878,172.343,28.986,155.337
C03120=1063.633,111.808,-75.898,172.345,28.989,155.338
C03121=1063.639,112.057,-75.917,172.346,28.992,155.338
C03122=1063.645,112.306,-75.937,172.348,28.994,155.338
C03123=1063.651,112.555,-75.956,172.350,28.997,155.339
C03124=1063.657,112.804,-75.976,172.351,29.000,155.339
C03125=1063.662,113.054,-75.995,172.353,29.002,155.340
C03126=1063.668,113.303,-76.015,172.354,29.005,155.340
C03127=1063.674,113.552,-76.034,172.355,29.008,155.341
C03128=1063.680,113.801,-76.054,172.357,29.010,155.341
C03129=1063.686,114.050,-76.074,172.358,29.013,155.341
C03130=1063.691,114.300,-76.093,172.360,29.016,155.342
C03131=1063.697,114.548,-76.113,172.362,29.019,155.342
C03132=1063.703,114.798,-76.132,172.363,29.021,155.343
C03133=1063.709,115.047,-76.152,172.365,29.024,155.343
C03134=1063.714,115.296,-76.172,172.367,29.027,155.343
C03135=1063.720,115.545,-76.192,172.368,29.030,155.344
C03136=1063.726,115.794,-76.212,172.370,29.032,155.344
C03137=1063.732,116.043,-76.231,172.372,29.035,155.345
C03138=1063.738,116.292,-76.251,172.373,29.038,155.345
C03139=1063.743,116.542,-76.270,172.375,29.041,155.346
C03140=1063.749,116.791,-76.291,172.376,29.044,155.346
C03141=1063.754,117.040,-76.310,172.378,29.047,155.346
C03142=1063.760,117.289,-76.330,172.380,29.049,155.347
C03143=1063.767,117.539,-76.350,172.381,29.052,155.347
C03144=1063.773,117.788,-76.370,172.382,29.055,155.348
C03145=1063.779,118.037,-76.389,172.384,29.057,155.348
C03146=1063.783,118.287,-76.409,172.385,29.060,155.348
C03147=1063.789,118.535,-76.429,172.387,29.063,155.349
C03148=1063.795,118.784,-76.449,172.389,29.066,155.349
C03149=1063.801,119.034,-76.468,172.390,29.068,155.350
C03150=1063.807,119.282,-76.488,172.392,29.071,155.350
C03151=1063.812,119.532,-76.509,172.394,29.074,155.350
C03152=1063.818,119.781,-76.528,172.395,29.077,155.351
C03153=1063.824,120.030,-76.548,172.397,29.079,155.351
C03154=1063.830,120.279,-76.568,172.398,29.082,155.352
C03155=1063.835,120.528,-76.588,172.400,29.085,155.352
C03156=1063.842,120.778,-76.608,172.402,29.087,155.352
C03157=1063.848,121.027,-76.628,172.403,29.090,155.353
C03158=1063.854,121.276,-76.648,172.405,29.093,155.353
C03159=1063.859,121.525,-76.667,172.407,29.096,155.354
C03160=1063.865,121.774,-76.688,172.408,29.098,155.354
C03161=1063.871,122.023,-76.708,172.410,29.101,155.354
C03162=1063.877,122.272,-76.728,172.412,29.104,155.355
C03163=1063.882,122.521,-76.747,172.413,29.107,155.355
C03164=1063.888,122.771,-76.768,172.415,29.110,155.356
C03165=1063.894,123.020,-76.788,172.417,29.113,155.356
C03166=1063.900,123.269,-76.808,172.418,29.115,155.357
C03167=1063.906,123.518,-76.827,172.420,29.118,155.357
C03168=1063.911,123.767,-76.848,172.421,29.121,155.357
C03169=1063.917,124.016,-76.868,172.423,29.124,155.358
C03170=1063.924,124.266,-76.888,172.425,29.126,155.358
C03171=1063.930,124.514,-76.908,172.427,29.128,155.359
C03172=1063.935,124.763,-76.929,172.428,29.131,155.359
C03173=1063.941,125.013,-76.948,172.430,29.134,155.359
C03174=1063.947,125.262,-76.968,172.431,29.137,155.360
C03175=1063.953,125.511,-76.988,172.433,29.139,155.360
C03176=1063.963,125.932,-77.022,172.436,29.144,155.361
C03177=1063.972,126.353,-77.056,172.438,29.149,155.362
C03178=1063.983,126.775,-77.090,172.441,29.154,155.362
C03179=1063.992,127.196,-77.124,172.444,29.158,155.363
C03180=1063.998,127.446,-77.145,172.445,29.160,155.363
C03181=1064.004,127.695,-77.165,172.447,29.163,155.364
C03182=1064.010,127.944,-77.185,172.449,29.166,155.364
C03183=1064.016,128.193,-77.205,172.450,29.169,155.365
C03184=1064.022,128.443,-77.226,172.452,29.171,155.365
C03185=1064.028,128.691,-77.246,172.454,29.174,155.365
C03186=1064.034,128.940,-77.266,172.455,29.177,155.366
C03187=1064.039,129.189,-77.286,172.457,29.179,155.366
C03188=1064.046,129.439,-77.307,172.459,29.182,155.367
C03189=1064.052,129.688,-77.327,172.460,29.185,155.367
C03190=1064.057,129.937,-77.347,172.462,29.188,155.367
C03191=1064.064,130.186,-77.368,172.464,29.190,155.368
C03192=1064.070,130.435,-77.388,172.465,29.193,155.368
C03193=1064.075,130.684,-77.408,172.467,29.196,155.369
C03194=1064.082,130.934,-77.428,172.469,29.198,155.369
C03195=1064.088,131.183,-77.448,172.470,29.201,155.369
C03196=1064.093,131.432,-77.469,172.472,29.203,155.370
C03197=1064.100,131.681,-77.489,172.474,29.206,155.370
C03198=1064.106,131.930,-77.509,172.475,29.209,155.370
C03199=1064.111,132.179,-77.531,172.477,29.212,155.371
C03200=1064.117,132.427,-77.551,172.479,29.214,155.371
C03201=1064.123,132.677,-77.571,172.480,29.217,155.372
C03202=1064.128,132.926,-77.592,172.482,29.220,155.372
C03203=1064.134,133.175,-77.612,172.484,29.223,155.373
C03204=1064.140,133.425,-77.633,172.486,29.226,155.373
C03205=1064.146,133.673,-77.654,172.488,29.229,155.373
C03206=1064.152,133.922,-77.674,172.489,29.231,155.374
C03207=1064.158,134.171,-77.694,172.491,29.234,155.374
C03208=1064.163,134.421,-77.715,172.493,29.237,155.375
C03209=1064.169,134.670,-77.736,172.494,29.240,155.375
C03210=1064.175,134.918,-77.756,172.496,29.242,155.375
C03211=1064.181,135.168,-77.777,172.498,29.245,155.376
C03212=1064.187,135.417,-77.797,172.499,29.248,155.376
C03213=1064.192,135.666,-77.818,172.501,29.250,155.377
C03214=1064.198,135.915,-77.839,172.503,29.253,155.377
C03215=1064.204,136.164,-77.859,172.504,29.256,155.377
C03216=1064.210,136.413,-77.880,172.506,29.259,155.378
C03217=1064.216,136.663,-77.900,172.508,29.261,155.378
C03218=1064.222,136.911,-77.921,172.509,29.264,155.379
C03219=1064.228,137.161,-77.942,172.511,29.267,155.379
C03220=1064.234,137.410,-77.962,172.513,29.269,155.380
C03221=1064.239,137.658,-77.984,172.514,29.272,155.380
C03222=1064.245,137.908,-78.004,172.516,29.275,155.380
C03223=1064.251,138.157,-78.024,172.518,29.278,155.381
C03224=1064.257,138.405,-78.046,172.519,29.280,155.381
C03225=1064.262,138.655,-78.067,172.521,29.283,155.382
C03226=1064.268,138.904,-78.087,172.523,29.286,155.382
C03227=1064.275,139.153,-78.108,172.524,29.289,155.383
C03228=1064.280,139.402,-78.129,172.527,29.292,155.383
C03229=1064.286,139.651,-78.149,172.529,29.295,155.383
C03230=1064.292,139.900,-78.170,172.530,29.297,155.384
C03231=1064.297,140.150,-78.191,172.532,29.300,155.384
C03232=1064.303,140.399,-78.213,172.534,29.303,155.385
C03233=1064.309,140.648,-78.232,172.535,29.306,155.385
C03234=1064.315,140.896,-78.254,172.537,29.308,155.385
C03235=1064.321,141.146,-78.275,172.539,29.311,155.386
C03236=1064.326,141.394,-78.296,172.540,29.314,155.386
C03237=1064.332,141.644,-78.317,172.542,29.316,155.387
C03238=1064.338,141.893,-78.338,172.544,29.319,155.387
C03239=1064.344,142.142,-78.358,172.545,29.322,155.387
C03240=1064.350,142.426,-78.382,172.548,29.325,155.388
C03241=1064.357,142.710,-78.406,172.549,29.329,155.388
C03242=1064.364,142.994,-78.430,172.551,29.332,155.389
C03243=1064.370,143.277,-78.454,172.554,29.335,155.389
C03244=1064.376,143.526,-78.475,172.555,29.338,155.390
C03245=1064.381,143.775,-78.496,172.557,29.340,155.390
C03246=1064.388,144.025,-78.518,172.559,29.343,155.391
C03247=1064.393,144.273,-78.539,172.560,29.346,155.391
C03248=1064.399,144.523,-78.560,172.562,29.349,155.391
C03249=1064.405,144.771,-78.580,172.564,29.352,155.392
C03250=1064.411,145.020,-78.601,172.565,29.354,155.392
C03251=1064.417,145.269,-78.623,172.567,29.357,155.393
C03252=1064.422,145.518,-78.644,172.569,29.360,155.393
C03253=1064.428,145.768,-78.665,172.571,29.363,155.393
C03254=1064.434,146.016,-78.686,172.573,29.365,155.394
C03255=1064.440,146.266,-78.707,172.575,29.368,155.394
C03256=1064.445,146.515,-78.728,172.576,29.371,155.395
C03257=1064.452,146.763,-78.749,172.578,29.374,155.395
C03258=1064.457,147.013,-78.770,172.580,29.376,155.396
C03259=1064.463,147.262,-78.791,172.581,29.379,155.396
C03260=1064.470,147.511,-78.813,172.583,29.382,155.396
C03261=1064.475,147.759,-78.834,172.585,29.384,155.397
C03262=1064.481,148.009,-78.855,172.586,29.387,155.397
C03263=1064.487,148.258,-78.877,172.589,29.391,155.398
C03264=1064.493,148.507,-78.898,172.591,29.393,155.398
C03265=1064.498,148.756,-78.919,172.592,29.396,155.398
C03266=1064.504,149.005,-78.940,172.594,29.399,155.399
C03267=1064.510,149.254,-78.962,172.596,29.401,155.399
C03268=1064.516,149.503,-78.983,172.597,29.404,155.400
C03269=1064.521,149.752,-79.005,172.599,29.407,155.400
C03270=1064.527,150.001,-79.025,172.601,29.410,155.401
C03271=1064.533,150.250,-79.047,172.602,29.413,155.401
C03272=1064.539,150.499,-79.068,172.605,29.416,155.401
C03273=1064.544,150.748,-79.090,172.607,29.418,155.402
C03274=1064.550,150.997,-79.112,172.608,29.421,155.402
C03275=1064.556,151.246,-79.133,172.610,29.424,155.403
C03276=1064.561,151.495,-79.154,172.612,29.427,155.403
C03277=1064.568,151.745,-79.176,172.613,29.429,155.403
C03278=1064.573,151.993,-79.197,172.615,29.433,155.404
C03279=1064.579,152.242,-79.219,172.617,29.435,155.404
C03280=1064.585,152.491,-79.240,172.619,29.438,155.405
C03281=1064.591,152.740,-79.262,172.621,29.441,155.405
C03282=1064.596,152.989,-79.283,172.623,29.444,155.406
C03283=1064.602,153.238,-79.305,172.624,29.446,155.406
C03284=1064.608,153.487,-79.327,172.626,29.449,155.406
C03285=1064.614,153.736,-79.348,172.628,29.452,155.407
C03286=1064.620,153.986,-79.369,172.629,29.455,155.407
C03287=1064.625,154.234,-79.390,172.632,29.458,155.408
C03288=1064.631,154.483,-79.412,172.634,29.461,155.408
C03289=1064.637,154.733,-79.434,172.635,29.463,155.409
C03290=1064.642,154.981,-79.455,172.637,29.466,155.409
C03291=1064.648,155.231,-79.477,172.639,29.469,155.409
C03292=1064.654,155.479,-79.498,172.640,29.471,155.410
C03293=1064.660,155.728,-79.520,172.642,29.475,155.410
C03294=1064.666,155.978,-79.542,172.645,29.478,155.411
C03295=1064.671,156.226,-79.563,172.646,29.480,155.411
C03296=1064.678,156.475,-79.586,172.648,29.483,155.412
C03297=1064.684,156.724,-79.607,172.650,29.486,155.412
C03298=1064.689,156.973,-79.629,172.651,29.488,155.412
C03299=1064.695,157.222,-79.651,172.653,29.492,155.413
C03300=1064.701,157.471,-79.672,172.656,29.494,155.413
C03301=1064.706,157.720,-79.694,172.657,29.497,155.414
C03302=1064.712,157.969,-79.716,172.659,29.500,155.414
C03303=1064.718,158.218,-79.737,172.661,29.503,155.415
C03304=1064.724,158.502,-79.762,172.663,29.506,155.415
C03305=1064.731,158.785,-79.787,172.665,29.509,155.416
C03306=1064.738,159.068,-79.812,172.667,29.512,155.416
C03307=1064.744,159.352,-79.837,172.669,29.515,155.416
C03308=1064.750,159.601,-79.859,172.671,29.518,155.417
C03309=1064.756,159.850,-79.880,172.672,29.521,155.417
C03310=1064.761,160.099,-79.902,172.675,29.524,155.418
C03311=1064.767,160.349,-79.924,172.677,29.527,155.418
C03312=1064.774,160.597,-79.946,172.678,29.530,155.419
C03313=1064.779,160.846,-79.968,172.680,29.532,155.419
C03314=1064.785,161.095,-79.990,172.682,29.535,155.419
C03315=1064.791,161.344,-80.012,172.683,29.538,155.420
C03316=1064.796,161.593,-80.034,172.686,29.541,155.420
C03317=1064.802,161.842,-80.056,172.688,29.544,155.421
C03318=1064.808,162.091,-80.078,172.689,29.547,155.421
C03319=1064.813,162.340,-80.100,172.691,29.550,155.422
C03320=1064.818,162.589,-80.123,172.693,29.553,155.422
C03321=1064.824,162.838,-80.144,172.695,29.556,155.423
C03322=1064.829,163.087,-80.166,172.697,29.559,155.423
C03323=1064.835,163.336,-80.189,172.699,29.561,155.423
C03324=1064.841,163.584,-80.210,172.700,29.565,155.424
C03325=1064.846,163.833,-80.233,172.702,29.567,155.424
C03326=1064.852,164.083,-80.256,172.705,29.570,155.425
C03327=1064.858,164.332,-80.277,172.706,29.574,155.425
C03328=1064.863,164.580,-80.300,172.708,29.576,155.426
C03329=1064.869,164.829,-80.322,172.710,29.579,155.426
C03330=1064.875,165.078,-80.344,172.711,29.582,155.427
C03331=1064.880,165.327,-80.366,172.714,29.585,155.427
C03332=1064.886,165.576,-80.388,172.716,29.588,155.427
C03333=1064.892,165.825,-80.411,172.717,29.591,155.428
C03334=1064.897,166.074,-80.433,172.719,29.594,155.428
C03335=1064.903,166.323,-80.455,172.721,29.596,155.429
C03336=1064.908,166.572,-80.477,172.723,29.600,155.429
C03337=1064.914,166.821,-80.500,172.725,29.603,155.430
C03338=1064.919,167.070,-80.522,172.727,29.605,155.430
C03339=1064.925,167.319,-80.544,172.728,29.608,155.431
C03340=1064.931,167.568,-80.567,172.730,29.611,155.431
C03341=1064.937,167.817,-80.590,172.733,29.614,155.431
C03342=1064.943,168.066,-80.611,172.734,29.617,155.432
C03343=1064.948,168.314,-80.634,172.736,29.620,155.432
C03344=1064.953,168.564,-80.656,172.738,29.623,155.433
C03345=1064.960,168.812,-80.678,172.740,29.626,155.433
C03346=1064.965,169.062,-80.701,172.742,29.629,155.434
C03347=1064.970,169.310,-80.723,172.744,29.632,155.434
C03348=1064.976,169.559,-80.746,172.745,29.634,155.435
C03349=1064.982,169.808,-80.768,172.748,29.638,155.435
C03350=1064.988,170.057,-80.791,172.750,29.640,155.435
C03351=1064.993,170.307,-80.813,172.751,29.643,155.436
C03352=1065.000,170.555,-80.835,172.753,29.646,155.436
C03353=1065.005,170.803,-80.858,172.756,29.649,155.437
C03354=1065.010,171.053,-80.880,172.757,29.652,155.437
C03355=1065.016,171.302,-80.903,172.759,29.655,155.438
C03356=1065.023,171.550,-80.925,172.761,29.658,155.438
C03357=1065.028,171.800,-80.948,172.763,29.661,155.439
C03358=1065.034,172.049,-80.971,172.765,29.663,155.439
C03359=1065.039,172.298,-80.994,172.767,29.667,155.439
C03360=1065.045,172.546,-81.016,172.768,29.669,155.440
C03361=1065.051,172.795,-81.038,172.771,29.672,155.440
C03362=1065.057,173.044,-81.061,172.773,29.676,155.441
C03363=1065.062,173.293,-81.084,172.774,29.678,155.441
C03364=1065.068,173.542,-81.105,172.777,29.681,155.442
C03365=1065.074,173.791,-81.128,172.779,29.684,155.442
C03366=1065.080,174.040,-81.151,172.780,29.687,155.443
C03367=1065.086,174.289,-81.174,172.782,29.690,155.443
C03368=1065.092,174.572,-81.200,172.785,29.693,155.443
C03369=1065.099,174.855,-81.225,172.787,29.697,155.444
C03370=1065.106,175.138,-81.251,172.789,29.700,155.445
C03371=1065.112,175.422,-81.277,172.792,29.703,155.445
C03372=1065.118,175.670,-81.300,172.793,29.706,155.445
C03373=1065.123,175.919,-81.323,172.795,29.709,155.446
C03374=1065.129,176.168,-81.345,172.798,29.712,155.446
C03375=1065.135,176.417,-81.367,172.799,29.715,155.447
C03376=1065.141,176.666,-81.390,172.801,29.717,155.447
C03377=1065.147,176.915,-81.413,172.804,29.720,155.448
C03378=1065.152,177.163,-81.436,172.805,29.724,155.448
C03379=1065.158,177.412,-81.459,172.807,29.726,155.449
C03380=1065.165,177.661,-81.481,172.810,29.729,155.449
C03381=1065.170,177.910,-81.504,172.811,29.732,155.449
C03382=1065.176,178.159,-81.527,172.813,29.735,155.450
C03383=1065.182,178.408,-81.550,172.815,29.738,155.450
C03384=1065.187,178.657,-81.572,172.817,29.741,155.451
C03385=1065.194,178.906,-81.595,172.819,29.744,155.451
C03386=1065.199,179.155,-81.618,172.821,29.747,155.452
C03387=1065.205,179.404,-81.641,172.824,29.749,155.452
C03388=1065.211,179.653,-81.664,172.825,29.752,155.452
C03389=1065.217,179.902,-81.687,172.827,29.755,155.453
C03390=1065.223,180.151,-81.710,172.830,29.758,155.453
C03391=1065.229,180.400,-81.732,172.831,29.761,155.454
C03392=1065.235,180.648,-81.755,172.833,29.764,155.454
C03393=1065.241,180.897,-81.778,172.836,29.767,155.455
C03394=1065.247,181.146,-81.802,172.837,29.770,155.455
C03395=1065.253,181.394,-81.825,172.840,29.773,155.455
C03396=1065.258,181.643,-81.848,172.842,29.776,155.456
C03397=1065.264,181.892,-81.870,172.843,29.778,155.456
C03398=1065.271,182.141,-81.893,172.846,29.781,155.457
C03399=1065.276,182.390,-81.916,172.848,29.784,155.457
C03400=1065.283,182.639,-81.939,172.849,29.787,155.458
C03401=1065.288,182.888,-81.962,172.852,29.790,155.458
C03402=1065.294,183.137,-81.985,172.854,29.793,155.459
C03403=1065.300,183.386,-82.008,172.855,29.796,155.459
C03404=1065.306,183.634,-82.032,172.858,29.799,155.460
C03405=1065.312,183.883,-82.055,172.860,29.802,155.460
C03406=1065.318,184.132,-82.077,172.862,29.804,155.460
C03407=1065.324,184.381,-82.100,172.864,29.808,155.461
C03408=1065.330,184.630,-82.123,172.866,29.810,155.461
C03409=1065.335,184.879,-82.147,172.868,29.814,155.462
C03410=1065.341,185.128,-82.170,172.870,29.816,155.462
C03411=1065.347,185.377,-82.193,172.872,29.820,155.463
C03412=1065.352,185.626,-82.217,172.875,29.823,155.463
C03413=1065.358,185.874,-82.241,172.876,29.826,155.464
C03414=1065.364,186.123,-82.263,172.878,29.828,155.464
C03415=1065.369,186.372,-82.287,172.881,29.832,155.465
C03416=1065.375,186.621,-82.311,172.882,29.835,155.465
C03417=1065.380,186.869,-82.334,172.885,29.838,155.465
C03418=1065.385,187.119,-82.357,172.887,29.841,155.466
C03419=1065.391,187.367,-82.381,172.888,29.844,155.466
C03420=1065.397,187.616,-82.404,172.891,29.847,155.467
C03421=1065.402,187.865,-82.427,172.893,29.850,155.467
C03422=1065.409,188.114,-82.451,172.894,29.853,155.468
C03423=1065.414,188.363,-82.474,172.897,29.856,155.468
C03424=1065.420,188.612,-82.499,172.899,29.859,155.469
C03425=1065.426,188.860,-82.521,172.901,29.863,155.469
C03426=1065.431,189.109,-82.544,172.903,29.865,155.470
C03427=1065.437,189.358,-82.569,172.905,29.869,155.470
C03428=1065.442,189.607,-82.592,172.907,29.872,155.471
C03429=1065.448,189.855,-82.616,172.909,29.875,155.471
C03430=1065.454,190.105,-82.639,172.912,29.878,155.472
C03431=1065.460,190.353,-82.663,172.913,29.881,155.472
C03432=1065.466,190.636,-82.690,172.916,29.884,155.473
C03433=1065.473,190.919,-82.716,172.918,29.887,155.473
C03434=1065.479,191.202,-82.744,172.920,29.891,155.474
C03435=1065.486,191.484,-82.770,172.923,29.895,155.474
C03436=1065.491,191.734,-82.794,172.925,29.898,155.475
C03437=1065.497,191.982,-82.817,172.927,29.901,155.475
C03438=1065.503,192.231,-82.840,172.929,29.904,155.476
C03439=1065.508,192.479,-82.865,172.932,29.907,155.476
C03440=1065.514,192.728,-82.889,172.933,29.910,155.477
C03441=1065.519,192.978,-82.912,172.935,29.913,155.477
C03442=1065.525,193.226,-82.936,172.938,29.916,155.478
C03443=1065.531,193.475,-82.959,172.939,29.919,155.478
C03444=1065.537,193.724,-82.983,172.942,29.922,155.479
C03445=1065.543,193.972,-83.007,172.944,29.925,155.479
C03446=1065.548,194.222,-83.031,172.946,29.929,155.480
C03447=1065.554,194.470,-83.054,172.948,29.932,155.480
C03448=1065.560,194.719,-83.079,172.951,29.935,155.480
C03449=1065.566,194.968,-83.102,172.952,29.938,155.481
C03450=1065.572,195.216,-83.126,172.954,29.941,155.481
C03451=1065.577,195.465,-83.150,172.957,29.944,155.482
C03452=1065.583,195.714,-83.173,172.958,29.947,155.482
C03453=1065.589,195.963,-83.197,172.961,29.950,155.483
C03454=1065.595,196.211,-83.221,172.963,29.953,155.483
C03455=1065.601,196.461,-83.246,172.965,29.956,155.484
C03456=1065.606,196.710,-83.269,172.967,29.959,155.484
C03457=1065.612,196.958,-83.293,172.970,29.962,155.485
C03458=1065.618,197.207,-83.317,172.971,29.965,155.485
C03459=1065.624,197.456,-83.341,172.974,29.968,155.486
C03460=1065.630,197.704,-83.365,172.976,29.971,155.486
C03461=1065.635,197.954,-83.389,172.978,29.975,155.487
C03462=1065.641,198.202,-83.412,172.980,29.978,155.487
C03463=1065.647,198.450,-83.436,172.983,29.981,155.488
C03464=1065.653,198.700,-83.461,172.985,29.984,155.488
C03465=1065.659,198.948,-83.484,172.987,29.987,155.489
C03466=1065.665,199.197,-83.509,172.989,29.990,155.489
C03467=1065.671,199.446,-83.532,172.992,29.993,155.489
C03468=1065.676,199.695,-83.556,172.993,29.996,155.490
C03469=1065.683,199.944,-83.580,172.996,29.999,155.490
C03470=1065.688,200.192,-83.604,172.998,30.002,155.491
C03471=1065.694,200.441,-83.628,173.000,30.006,155.491
C03472=1065.700,200.690,-83.653,173.002,30.008,155.492
C03473=1065.706,200.938,-83.676,173.005,30.012,155.492
C03474=1065.712,201.187,-83.701,173.006,30.014,155.493
C03475=1065.717,201.436,-83.725,173.009,30.018,155.493
C03476=1065.723,201.684,-83.749,173.011,30.021,155.494
C03477=1065.729,201.934,-83.774,173.013,30.024,155.494
C03478=1065.735,202.182,-83.797,173.015,30.027,155.495
C03479=1065.741,202.431,-83.822,173.018,30.031,155.495
C03480=1065.747,202.680,-83.846,173.019,30.033,155.496
C03481=1065.753,202.928,-83.870,173.022,30.037,155.496
C03482=1065.758,203.177,-83.894,173.024,30.040,155.497
C03483=1065.764,203.426,-83.919,173.026,30.043,155.497
C03484=1065.770,203.675,-83.943,173.028,30.046,155.498
C03485=1065.775,203.924,-83.968,173.031,30.049,155.498
C03486=1065.781,204.172,-83.991,173.033,30.053,155.499
C03487=1065.787,204.421,-84.017,173.035,30.056,155.499
C03488=1065.793,204.669,-84.041,173.037,30.059,155.500
C03489=1065.798,204.919,-84.065,173.040,30.062,155.500
C03490=1065.804,205.167,-84.090,173.042,30.065,155.501
C03491=1065.810,205.416,-84.114,173.044,30.069,155.501
C03492=1065.816,205.665,-84.138,173.047,30.072,155.502
C03493=1065.822,205.913,-84.163,173.048,30.075,155.502
C03494=1065.827,206.162,-84.188,173.051,30.078,155.503
C03495=1065.833,206.411,-84.212,173.053,30.081,155.503
C03496=1065.857,207.456,-84.315,173.209,30.159,155.508
C03497=1065.863,207.676,-84.337,173.211,30.163,155.509
C03498=1065.868,207.897,-84.359,173.213,30.166,155.510
C03499=1065.874,208.116,-84.382,173.214,30.170,155.510
C03500=1065.879,208.336,-84.404,173.216,30.173,155.511
C03501=1065.884,208.556,-84.426,173.218,30.177,155.512
C03502=1065.889,208.776,-84.449,173.219,30.181,155.512
C03503=1065.894,208.995,-84.472,173.221,30.184,155.513
C03504=1065.900,209.215,-84.494,173.223,30.188,155.513
C03505=1065.905,209.464,-84.519,173.225,30.192,155.514
C03506=1065.911,209.712,-84.544,173.227,30.196,155.515
C03507=1065.917,209.961,-84.569,173.229,30.200,155.516
C03508=1065.923,210.210,-84.595,173.231,30.204,155.516
C03509=1065.930,210.458,-84.620,173.233,30.208,155.517
C03510=1065.936,210.707,-84.645,173.234,30.212,155.518
C03511=1065.941,210.956,-84.671,173.237,30.216,155.518
C03512=1065.948,211.205,-84.697,173.239,30.221,155.519
C03513=1065.953,211.453,-84.722,173.240,30.224,155.520
C03514=1065.960,211.701,-84.748,173.243,30.229,155.521
C03515=1065.965,211.950,-84.774,173.245,30.233,155.521
C03516=1065.971,212.198,-84.799,173.247,30.237,155.522
C03517=1065.978,212.447,-84.824,173.249,30.241,155.523
C03518=1065.983,212.696,-84.850,173.250,30.245,155.523
C03519=1065.989,212.945,-84.876,173.253,30.249,155.524
C03520=1065.995,213.193,-84.901,173.255,30.253,155.525
C03521=1066.001,213.442,-84.927,173.256,30.257,155.526
C03522=1066.007,213.691,-84.952,173.259,30.261,155.526
C03523=1066.013,213.938,-84.978,173.261,30.265,155.527
C03524=1066.019,214.187,-85.004,173.263,30.269,155.528
C03525=1066.025,214.436,-85.029,173.265,30.274,155.528
C03526=1066.030,214.685,-85.055,173.266,30.277,155.529
C03527=1066.036,214.934,-85.080,173.269,30.282,155.530
C03528=1066.043,215.182,-85.106,173.271,30.286,155.531
C03529=1066.048,215.431,-85.132,173.272,30.290,155.531
C03530=1066.055,215.679,-85.158,173.275,30.294,155.532
C03531=1066.060,215.928,-85.184,173.277,30.298,155.533
C03532=1066.067,216.176,-85.210,173.279,30.302,155.533
C03533=1066.072,216.425,-85.236,173.281,30.306,155.534
C03534=1066.078,216.674,-85.261,173.282,30.310,155.535
C03535=1066.085,216.922,-85.287,173.285,30.314,155.535
C03536=1066.090,217.171,-85.313,173.287,30.318,155.536
C03537=1066.096,217.420,-85.338,173.289,30.322,155.537
C03538=1066.102,217.668,-85.365,173.291,30.327,155.538
C03539=1066.108,217.917,-85.390,173.294,30.330,155.538
C03540=1066.114,218.166,-85.416,173.295,30.334,155.539
C03541=1066.120,218.414,-85.442,173.297,30.339,155.540
C03542=1066.126,218.663,-85.468,173.300,30.342,155.540
C03543=1066.132,218.911,-85.493,173.301,30.347,155.541
C03544=1066.138,219.160,-85.520,173.304,30.351,155.542
C03545=1066.144,219.409,-85.545,173.306,30.354,155.542
C03546=1066.150,219.657,-85.572,173.307,30.359,155.543
C03547=1066.156,219.906,-85.597,173.310,30.363,155.544
C03548=1066.162,220.154,-85.624,173.312,30.366,155.545
C03549=1066.168,220.403,-85.649,173.314,30.371,155.545
C03550=1066.174,220.651,-85.676,173.316,30.375,155.546
C03551=1066.180,220.900,-85.701,173.318,30.378,155.547
C03552=1066.187,221.148,-85.728,173.320,30.383,155.547
C03553=1066.191,221.371,-85.751,173.322,30.386,155.548
C03554=1066.196,221.593,-85.774,173.323,30.390,155.549
C03555=1066.202,221.815,-85.798,173.326,30.394,155.549
C03556=1066.207,222.037,-85.821,173.328,30.397,155.550
C03557=1066.213,222.259,-85.844,173.330,30.401,155.551
C03558=1066.218,222.482,-85.868,173.331,30.404,155.551
C03559=1066.223,222.703,-85.891,173.333,30.408,155.552
C03560=1066.228,222.926,-85.915,173.336,30.412,155.552
C03561=1066.235,223.174,-85.941,173.337,30.416,155.553
C03562=1066.240,223.422,-85.967,173.339,30.420,155.554
C03563=1066.246,223.672,-85.994,173.342,30.424,155.555
C03564=1066.253,223.920,-86.020,173.343,30.428,155.555
C03565=1066.259,224.168,-86.046,173.346,30.432,155.556
C03566=1066.264,224.417,-86.072,173.347,30.436,155.557
C03567=1066.270,224.665,-86.099,173.350,30.440,155.557
C03568=1066.276,224.914,-86.125,173.352,30.444,155.558
C03569=1066.282,225.162,-86.151,173.354,30.448,155.559
C03570=1066.288,225.411,-86.178,173.356,30.452,155.560
C03571=1066.294,225.660,-86.205,173.359,30.456,155.560
C03572=1066.301,225.908,-86.231,173.360,30.460,155.561
C03573=1066.306,226.157,-86.257,173.363,30.464,155.562
C03574=1066.312,226.405,-86.283,173.365,30.468,155.562
C03575=1066.318,226.654,-86.310,173.367,30.472,155.563
C03576=1066.324,226.902,-86.336,173.369,30.476,155.564
C03577=1066.330,227.151,-86.362,173.372,30.480,155.564
C03578=1066.336,227.400,-86.389,173.373,30.484,155.565
C03579=1066.342,227.648,-86.416,173.376,30.488,155.566
C03580=1066.347,227.896,-86.442,173.378,30.492,155.566
C03581=1066.354,228.145,-86.468,173.379,30.496,155.567
C03582=1066.360,228.394,-86.495,173.382,30.500,155.568
C03583=1066.366,228.642,-86.522,173.384,30.504,155.569
C03584=1066.372,228.891,-86.548,173.386,30.508,155.569
C03585=1066.378,229.139,-86.574,173.389,30.512,155.570
C03586=1066.384,229.388,-86.601,173.391,30.516,155.571
C03587=1066.390,229.636,-86.628,173.393,30.520,155.571
C03588=1066.396,229.885,-86.654,173.395,30.524,155.572
C03589=1066.402,230.133,-86.681,173.398,30.528,155.573
C03590=1066.408,230.382,-86.708,173.399,30.532,155.573
C03591=1066.414,230.631,-86.734,173.402,30.536,155.574
C03592=1066.420,230.879,-86.761,173.404,30.540,155.575
C03593=1066.426,231.127,-86.788,173.406,30.544,155.575
C03594=1066.432,231.376,-86.815,173.408,30.548,155.576
C03595=1066.438,231.625,-86.841,173.411,30.552,155.577
C03596=1066.443,231.873,-86.868,173.412,30.556,155.578
C03597=1066.449,232.121,-86.895,173.415,30.560,155.578
C03598=1066.456,232.370,-86.922,173.417,30.564,155.579
C03599=1066.461,232.619,-86.948,173.419,30.568,155.580
C03600=1066.467,232.867,-86.975,173.421,30.572,155.580
C03601=1066.474,233.116,-87.003,173.424,30.576,155.581
C03602=1066.480,233.364,-87.029,173.425,30.580,155.582
C03603=1066.485,233.612,-87.056,173.428,30.584,155.583
C03604=1066.491,233.861,-87.083,173.430,30.588,155.583
C03605=1066.497,234.110,-87.110,173.432,30.592,155.584
C03606=1066.503,234.358,-87.136,173.434,30.596,155.585
C03607=1066.509,234.606,-87.164,173.437,30.600,155.585
C03608=1066.515,234.855,-87.191,173.439,30.604,155.586
C03609=1066.520,235.074,-87.214,173.441,30.608,155.587
C03610=1066.525,235.292,-87.238,173.443,30.611,155.587
C03611=1066.531,235.509,-87.262,173.445,30.614,155.588
C03612=1066.536,235.727,-87.286,173.446,30.618,155.589
C03613=1066.541,235.946,-87.309,173.449,30.621,155.589
C03614=1066.547,236.164,-87.333,173.451,30.625,155.590
C03615=1066.552,236.381,-87.357,173.453,30.629,155.590
C03616=1066.556,236.600,-87.381,173.454,30.632,155.591
C03617=1066.562,236.848,-87.408,173.457,30.636,155.592
C03618=1066.569,237.097,-87.435,173.460,30.640,155.592
C03619=1066.575,237.345,-87.462,173.461,30.644,155.593
C03620=1066.581,237.594,-87.489,173.464,30.648,155.594
C03621=1066.587,237.842,-87.516,173.466,30.652,155.594
C03622=1066.592,238.090,-87.544,173.468,30.656,155.595
C03623=1066.599,238.339,-87.571,173.470,30.660,155.596
C03624=1066.604,238.588,-87.597,173.473,30.664,155.597
C03625=1066.611,238.836,-87.625,173.475,30.668,155.597
C03626=1066.617,239.084,-87.652,173.477,30.672,155.598
C03627=1066.622,239.332,-87.680,173.480,30.676,155.599
C03628=1066.629,239.582,-87.707,173.482,30.680,155.599
C03629=1066.635,239.829,-87.734,173.484,30.684,155.600
C03630=1066.641,240.078,-87.761,173.487,30.688,155.601
C03631=1066.646,240.326,-87.789,173.489,30.692,155.601
C03632=1066.653,240.575,-87.816,173.491,30.696,155.602
C03633=1066.659,240.823,-87.844,173.493,30.700,155.603
C03634=1066.665,241.072,-87.871,173.496,30.703,155.603
C03635=1066.670,241.320,-87.899,173.498,30.708,155.604
